// TwinCAT 3 PLC project Welding_Robot_Control_Test
// ProgramVersion: 3.1.4020.4
// libraries:
//   Tc2_MC2, * (Beckhoff Automation GmbH)
//   Tc2_Standard, * (Beckhoff Automation GmbH)
//   Tc2_System, * (Beckhoff Automation GmbH)
//   Tc3_Module, * (Beckhoff Automation GmbH)
//   VisuDialogs, * (System)
// project tree:
//   DUTs/Axis/ Axis.TcPOU (not stored)
//   DUTs/Delay/ Delay.TcPOU (not stored)
//   DUTs/Filter_Current/ E_TcMatSimDataAreaType_1.TcDUT (not stored), FB_Filter_Current_Hexapod_Robot.TcPOU (not stored), FB_TcMatSimObject_1.TcPOU (not stored), ST_Filter_Current_Hexapod_Robot_InitData.TcDUT (not stored), ST_Filter_Current_Hexapod_Robot_Input.TcDUT (not stored), ST_Filter_Current_Hexapod_Robot_Output.TcDUT (not stored), ST_TcMatSimObjectDataAreaInfo_1.TcDUT (not stored)
//   DUTs/Hexapod_Leg/ Hexapod_Leg.TcPOU (not stored)
//   DUTs/Mapping/ Hexapod_Robot_Mapping.TcPOU (not stored)
//   DUTs/Robot_Simulink/ E_TcMatSimDataAreaType.TcDUT, FB_TcMatSimObject.TcPOU, FB_Welding_Control_Circle_86s.TcPOU, ST_TcMatSimObjectDataAreaInfo.TcDUT, ST_Welding_Control_Circle_86s_InitData.TcDUT, ST_Welding_Control_Circle_86s_Input.TcDUT, ST_Welding_Control_Circle_86s_Output.TcDUT
//   / GlobalTextList.TcGTLO, HexRobot_Task.TcTTO, PlcTask.TcTTO, Welding_Arm_Task.TcTTO, 视图管理器.TcVMO (not stored)
//   GVLs/ GVL.TcGVL
//   POUs/ Hexapod_Robot.TcPOU, Welding_Arm.TcPOU, Welding_Robot.TcPOU
//   VISUs/ Visu_Home.TcVIS, Visu_SimulinkMove.TcVIS, Visu_Power.TcVIS, Visu_Reset.TcVIS, Visu_Stand.TcVIS (not stored)

CONFIGURATION Welding_Robot_Control_Test
    RESOURCE PLC ON TwinCAT3
        TASK HexRobot_Task(INTERVAL := T#1ms, PRIORITY := 21);
        TASK PlcTask(INTERVAL := T#1ms, PRIORITY := 20);
        TASK Welding_Arm_Task(INTERVAL := T#1ms, PRIORITY := 22);
        PROGRAM Hexapod_Robot WITH HexRobot_Task : Hexapod_Robot;
        PROGRAM Welding_Robot WITH PlcTask : Welding_Robot;
        PROGRAM Welding_Arm WITH Welding_Arm_Task : Welding_Arm;
    END_RESOURCE
END_CONFIGURATION

// ---- DUTs/Robot_Simulink/E_TcMatSimDataAreaType.TcDUT
TYPE E_TcMatSimDataAreaType :
(
	NotSpecified := 0,
	Standard,
	InputSrc,
	InputDst,
	OutputSrc,
	OutputDst,
	InternalDa,
	MArea,
	RetainDa
);
END_TYPE

// ---- DUTs/Robot_Simulink/ST_TcMatSimObjectDataAreaInfo.TcDUT
TYPE ST_TcMatSimObjectDataAreaInfo :
STRUCT
	pPlcVar: PVOID;
	pModuleProcImg: PVOID;
	nSize: UDINT;
	nDataAreaId: UDINT;
	eDataAreaType: E_TcMatSimDataAreaType;
END_STRUCT
END_TYPE

// ---- DUTs/Robot_Simulink/ST_Welding_Control_Circle_86s_InitData.TcDUT
{attribute 'pack_mode' := '4'}
TYPE ST_Welding_Control_Circle_86s_InitData :
STRUCT
	Header: TComInitDataHdr;
	CallByHdr: TComInitDataElmHdr;
	CallBy: TctModuleCallByType;
	ExecutionSequenceHdr: TComInitDataElmHdr;
	ExecutionSequence: TctModuleExecutionSequenceType;
	StepSizeHdr: TComInitDataElmHdr;
	StepSize: TctStepSizeType;
	ExecuteModelCodeHdr: TComInitDataElmHdr;
	ExecuteModelCode: BOOL;
	ContextInfoArr_0_TaskOidHdr: TComInitDataElmHdr;
	ContextInfoArr_0_TaskOid: OTCID;
	ContextInfoArr_0_TaskPriorityHdr: TComInitDataElmHdr;
	ContextInfoArr_0_TaskPriority: UDINT;
	ContextInfoArr_0_TaskCycleTimeNsHdr: TComInitDataElmHdr;
	ContextInfoArr_0_TaskCycleTimeNs: UDINT;
	ContextInfoArr_0_TaskPortHdr: TComInitDataElmHdr;
	ContextInfoArr_0_TaskPort: UINT;
	ContextInfoArr_0_TaskSortOrderHdr: TComInitDataElmHdr;
	ContextInfoArr_0_TaskSortOrder: UDINT;
END_STRUCT
END_TYPE

// ---- DUTs/Robot_Simulink/ST_Welding_Control_Circle_86s_Input.TcDUT
TYPE ST_Welding_Control_Circle_86s_Input :
STRUCT
	t: LREAL;
END_STRUCT
END_TYPE

// ---- DUTs/Robot_Simulink/ST_Welding_Control_Circle_86s_Output.TcDUT
TYPE ST_Welding_Control_Circle_86s_Output :
STRUCT
	Disp_P: matrix_18_real_T;
END_STRUCT
END_TYPE

// ---- GVLs/GVL.TcGVL
VAR_GLOBAL
	Power_Execute 		: BOOL;							// 上电使能控制信号
	Home_Execute		: BOOL;							// 设置零点程序使能
	Reset_Execute		: BOOL;							// 电机驱动重置动作发生使能
	ExSetPoint_Execute	: BOOL;							// 机器人外部信号发生使能
	
	// ====================Simulink模块相关=====================
	Robot_Simulink		: FB_Welding_Control_Circle_86s(oid:=16#01010020);	// Simulink模型定义
	T_ALL				: LREAL:=100;						// Simulink模型运动总时长
	t_Interval			: LREAL:=0.001;						// 取样时间间隔，默认为1ms
	t					: LREAL:=0;							// 取样当前时间变量，以0为起点
	
	Filter_Current  : FB_Filter_Current_Hexapod_Robot(oid:=16#01010030);

END_VAR

// ---- POUs/Hexapod_Robot.TcPOU
PROGRAM Hexapod_Robot
VAR
// =======================NC轴变量==========================
	//Leg_Robot			: ARRAY[1..6] OF Hexapod_Leg;	// 定义六足的腿
	Axis_Robot			: ARRAY[1..18] OF Axis;			// 定义六足轴参量(可以调整数据上限来调整电机数目)
	//Axis_Delay			: Delay;						// 延迟程序
	Leg_Number			: INT;							// 定义机器人腿数
	Axis_Number 		: INT;							// 定义轴数目
	
	// ===================模块动作信号(按动作先后排列)==========
	Axis_Power			: ARRAY[1..18] OF BOOL;			// 单电机使能
	Robot_Power			: BOOL;							// 机器人所有电机使能
	
	Leg_Home_Set		: ARRAY[1..6] OF BOOL;	
	Axis_Home_Set		: ARRAY[1..18] OF BOOL;			// 单电机设定零点信号
	Robot_Home_Set		: BOOL;							// 机器人所有电机设定零点信号
	
	Move_Execute		: BOOL;							// 绝对运动使能信号
	Robot_Stand_Execute	: BOOL;							// 机器人站立程序使能	
	Axis_Absolute_Eable	: ARRAY[1..18] OF BOOL;			// 单电机绝对运动使能信号
	Robot_Absolute_Eable: ARRAY[1..18] OF BOOL;			// 机器人站立使能信号
	Axis_Move_Position	: ARRAY[1..18] OF LREAL;		// 电机绝对运动位置			
	
	ExtSetPointEnable	: BOOL;							// 外部信号发生信号
	ExtSetPointDisable	: BOOL;							// 外部信号结束信号
	
	Axis_Reset			: ARRAY[1..18] OF BOOL;			// 单电机驱动重置信号使能
	Robot_Reset			: BOOL;							// 机器人整体电机驱动重置
	Axis_ResetDone		: ARRAY[1..18] OF BOOL;			// 单电机驱动重置完成
	
	// ===================状态监测变量=======================
	Power_Status	: ARRAY[1..18] OF BOOL;				// 上电监测信号
	Leg_Home_Done	: ARRAY[1..6] OF BOOL;
	Home_Done		: ARRAY[1..18] OF BOOL;				// 找零监测信号
	MoveAbsoluteDone: ARRAY[1..18] OF BOOL;				// 电机运动监测信号
	
	Robot_Error		: BOOL;								// 机器人电机错误信号
	Axis_Error		: ARRAY[1..18] OF BOOL;				// 电机错误监测信号
	Axis_ErrorID	: ARRAY[1..18] OF UDINT;			// 电机错误号码监测信号
	
	Axis_ActPostion	: ARRAY[1..18] OF LREAL;			// 电机轴实际位置
	Difference_Position	: ARRAY[1..18] OF LREAL;		// 实际位置与输入位置差值
	
	// =======================模块中间变量======================
	//HomeDone_Number	: LREAL :=0;					//完成找零的轴数
	//ExSetPoint_Position	: ARRAY[1..18] OF LREAL;		// 外部信号位置
	//t					: LREAL :=0;
	
	// =======================驱动器信号监测====================
	Current_Turque_Value  AT%IW0 : ARRAY[1..18] OF INT ;	//电流、力矩相关值
	Max_Turque_Value 	: INT ;							// 设置最大力矩边界值
	
	// ====================Simulink模块相关=====================
	Mapping				: Hexapod_Robot_Mapping;			// 变量映射	
	Model_Position		: ARRAY[1..18] OF LREAL;			// Simulink中各个腿的位置
	ExSetPoint_Position	: ARRAY[1..18] OF LREAL;			// 外部信号位置		
	Home_Position 		: ARRAY[1..18] OF LREAL;			// Home结束后的位移值
	
	Current_Turque_Filter  : ARRAY[1..18] OF LREAL;			// 滤波后的电流值
 
END_VAR

// =======================子程序使能(永久运行)===================
Variable_Monitor();			// 变量监测子程序使能
Logic_Control();			// 逻辑控制子程序使能
Variable_Set();				// 各动作速度子程序使能
SetGenerator();				// 外部信号发生子程序使能
Leg_Action();				// 单腿运动子程序使能
Robot_Action();				// 机器人整体运动子程序使能

// =====================电机驱动重置=============================
IF Reset_Execute THEN
	FOR Axis_Number := 1 TO 18 {BY 1} DO
		Axis_Robot[Axis_Number].Reset(Drive_Reset:= Axis_Reset[Axis_Number]);
	END_FOR
END_IF

// =======================电机上电===============================
IF Power_Execute THEN
	Filter_Current.Execute();
	FOR Axis_Number := 1 TO 18 {BY 1} DO
		Axis_Robot[Axis_Number].Power(Axis_Enable:= Axis_Power[Axis_Number]);
	END_FOR
END_IF

// =======================找零程序===============================
IF Home_Execute THEN
	Robot_Simulink.Execute();	// Simulink模型使能，用来为找零后的电机提供初始位移
	FOR Axis_Number := 1 TO 18 {BY 1} DO
		Axis_Robot[Axis_Number].Home(Drive_Home:= Axis_Home_Set[Axis_Number]);
	END_FOR
END_IF

// =======================站立程序===============================
IF Move_Execute THEN
	FOR Axis_Number := 1 TO 18 {BY 1} DO
		Axis_Robot[Axis_Number].Move_Absolute(	Drive_Move_Absolute:= Axis_Absolute_Eable[Axis_Number], 
												Absolute_Position:= Axis_Move_Position[Axis_Number]);
	END_FOR
END_IF
	
// =======================外部信号运动程序=======================
IF ExSetPoint_Execute THEN
	//SetGenerator();			// 使能外部信号发生子程序
	Robot_Simulink.Execute();	// Simulink模型使能
	FOR Axis_Number := 1 TO 18 {BY 1} DO
		Axis_Robot[Axis_Number].ExtSetPoint(Drive_ExtSetPointEnable:= ExtSetPointEnable, 
											Drive_ExtSetPointDisable:= ExtSetPointDisable, 
											ExSetPosition:= ExSetPoint_Position[Axis_Number]);
	END_FOR
END_IF

ACTION Leg_Action:
// ===================机器人单挑腿找零程序====================
IF Home_Execute THEN
	FOR Leg_Number := 1 TO 6 {BY 1} DO
		IF Leg_Home_Set[Leg_Number] THEN		// 在可视化中，Leg_Home_Set为点动
			Axis_Home_Set[1+(Leg_Number-1)*3] := Leg_Home_Set[Leg_Number];
			Axis_Home_Set[2+(Leg_Number-1)*3] := Leg_Home_Set[Leg_Number];
			Axis_Home_Set[3+(Leg_Number-1)*3] := Leg_Home_Set[Leg_Number];
		ELSIF Home_Done[1+(Leg_Number-1)*3] AND Axis_Home_Set[2+(Leg_Number-1)*3] AND Axis_Home_Set[3+(Leg_Number-1)*3] THEN
			Leg_Home_Set[Leg_Number] := FALSE; 
		END_IF
	END_FOR
END_IF
END_ACTION

ACTION Logic_Control:
// =======================控制逻辑区==========================
// 保证所有的动作拥有合理的先后顺序，优化控制逻辑
// 也防止出现两个或两个以上动作同时进行的情况，保证控制安全

// ===================电机驱动重置逻辑========================
//FOR Axis_Number := 1 TO 18 {BY 1} DO
IF Axis_Error[1] OR Axis_Error[2] OR Axis_Error[3] OR Axis_Error[4] OR Axis_Error[5] OR Axis_Error[6]
	 OR Axis_Error[7] OR Axis_Error[8] OR Axis_Error[9] OR Axis_Error[10] OR Axis_Error[11] OR Axis_Error[12]
		OR Axis_Error[13] OR Axis_Error[14] OR Axis_Error[15] OR Axis_Error[16] OR Axis_Error[17] OR Axis_Error[18]
THEN
	Robot_Error := TRUE;
ELSE
	Robot_Error := FALSE;
END_IF
//END_FOR

IF Robot_Error THEN
	Reset_Execute := TRUE;
ELSIF NOT Robot_Error AND NOT Welding_Arm.Arm_Error THEN
	Reset_Execute := FALSE;
ELSIF NOT Reset_Execute THEN
	Axis_Reset[Axis_Number] := FALSE;
	Axis_Robot[Axis_Number].Reset(Drive_Reset:= Axis_Reset[Axis_Number]);
END_IF

// =====================上电程序逻辑==========================
IF NOT Power_Execute THEN
	FOR Axis_Number := 1 TO 18 {BY 1} DO
		Axis_Power[Axis_Number] := FALSE;
		Axis_Robot[Axis_Number].Power(Axis_Enable:= Axis_Power[Axis_Number]);
	END_FOR
END_IF

// =====================找零程序逻辑==========================
IF Home_Execute THEN
	FOR Axis_Number := 1 TO 18 {BY 1} DO
		IF Home_Done[Axis_Number] THEN			// 	丝杠到达零点位置后，单电j机标零使能位关闭			
			Axis_Home_Set[Axis_Number] :=0;	
			Axis_Robot[Axis_Number].Home(Drive_Home:= Axis_Home_Set[Axis_Number]);
		END_IF
	END_FOR
	Move_Execute :=0;							// 设定零点时，不能进行其他运动
	ExSetPoint_Execute :=0;
ELSIF NOT Home_Execute THEN
	FOR Axis_Number := 1 TO 18 {BY 1} DO
		//Axis_Start_Back[Axis_Number] :=0;
		Axis_Home_Set[Axis_Number] := 0;
	END_FOR
END_IF

// =====================机器人站立逻辑==========================
IF Move_Execute THEN
	//Absolute_Eable := TRUE;
	Home_Execute := FALSE;						// 站立运动使能时，机器人调零必须结束
	ExSetPoint_Execute :=0;						// 站立运动时，不能进行其他运动
	FOR Axis_Number := 1 TO 18 {BY 1} DO
		IF MoveAbsoluteDone[Axis_Number] THEN	// 	丝杠到达设定位置后，单电机绝对运动使能位关闭
			Axis_Absolute_Eable[Axis_Number] := FALSE;
		END_IF
	END_FOR
ELSIF NOT Move_Execute THEN						// 站立运动不使能,轴不能运动
	FOR Axis_Number := 1 TO 18 {BY 1} DO
		Axis_Absolute_Eable[Axis_Number] := FALSE;
		Axis_Robot[Axis_Number].Move_Absolute(	Drive_Move_Absolute:= Axis_Absolute_Eable[Axis_Number], 
												Absolute_Position:= Axis_Move_Position[Axis_Number]);
	END_FOR
END_IF

// =====================外部信号发生逻辑========================
IF ExSetPoint_Execute THEN
	Home_Execute := FALSE;						// 外部信号发生使能时，机器人调零必须结束
	Move_Execute :=0;							// 外部信号发生时，不能进行其他运动
ELSIF NOT ExSetPoint_Execute THEN
	ExtSetPointEnable := 0;						// 外部信号发生不使能时，外部信号不能进入程序
	ExtSetPointDisable :=0;
ELSIF ExtSetPointDisable THEN
	ExtSetPointEnable :=0;						// 外部信号发生停止与外部信号发生开始不能同时进行
END_IF
END_ACTION

ACTION Robot_Action:
// =================机器人整体运动命令区======================
// 六足所有电机整体控制

// ====================机器人驱动重置=========================
IF Robot_Reset THEN
	IF Reset_Execute THEN
		Axis_Reset[Axis_Number] := TRUE;
		FOR Axis_Number := 1 TO 18 {BY 1} DO
			Axis_Robot[Axis_Number].Reset(Drive_Reset:= Axis_Reset[Axis_Number]);
		END_FOR
	END_IF
END_IF	

// ===================机器人所有电机上电======================
IF Robot_Power THEN	
	IF Power_Execute THEN
		FOR Axis_Number := 1 TO 18 {BY 1} DO
			Axis_Power[Axis_Number] := TRUE ;
		END_FOR
	END_IF
END_IF
	
// ===================机器人找零程序=======================
IF Robot_Home_Set THEN				// 标零程序
	//Robot_Start_Back := FALSE;
	IF Home_Execute THEN
		Leg_Home_Set[3] := Leg_Home_Set[5] := Leg_Home_Set[1];	// 在整机调零时，1\3\5三条腿同时调零；
		Leg_Home_Set[4] := Leg_Home_Set[6] := Leg_Home_Set[2];	// 在整机调零时，2\4\6三条腿同时调零；
	ELSIF NOT Home_Execute THEN
		FOR Leg_Number := 1 TO 6 {BY 1} DO
			Leg_Home_Set[Leg_Number] := FALSE;
		END_FOR
	END_IF
ELSIF NOT Robot_Home_Set AND NOT Home_Execute THEN
	FOR Axis_Number := 1 TO 18 {BY 1} DO
	Axis_Home_Set[Axis_Number] := FALSE;
	END_FOR
END_IF

// =====================站立程序===============================
IF Robot_Stand_Execute THEN
	IF Move_Execute THEN
		FOR Axis_Number := 1 TO 18 {BY 1} DO
			IF MoveAbsoluteDone[Axis_Number] THEN		// 	丝杠到达设定位置后，单电机绝对运动使能位关闭
				Axis_Absolute_Eable[Axis_Number] := FALSE;
			ELSE
				Axis_Absolute_Eable[Axis_Number] := TRUE;
			END_IF
		END_FOR
	END_IF
ELSIF NOT Robot_Stand_Execute AND NOT Move_Execute THEN 
	FOR Axis_Number := 1 TO 18 {BY 1} DO
		Axis_Absolute_Eable[Axis_Number] := FALSE;
	END_FOR
END_IF

// ======================外部信号发生=========================
IF ExtSetPointEnable THEN	
	//FOR Axis_Number := 1 TO 2 {BY 1} DO
	t := t + t_Interval;
	ExtSetPointDisable := FALSE;
	//END_FOR
END_IF

IF t=0 THEN
	FOR Axis_Number := 1 TO 18 {BY 1} DO
		Home_Position[Axis_Number] := Axis_ActPostion[Axis_Number];
	END_FOR
ELSIF t>=T_ALL THEN
	ExtSetPointEnable := FALSE;
	t:=0;
	ExtSetPointDisable := TRUE;
END_IF
END_ACTION

ACTION SetGenerator:
// ====================外部信号发生测试区=====================
// 用来测试外部信号发生功能和电机相关参数

// =================外部信号正弦信号发生======================
(*IF ExtSetPointEnable THEN
	FOR Axis_Number := 1 TO 18 {BY 1} DO
		ExSetPoint_Position[Axis_Number]:=10*SIN(2*3.14*t);
		t := t+0.001;
	END_FOR
END_IF

// =================外部信号停止逻辑判断=======================
//IF Axis_Robot[Axis_Number].State_ExtSetPiontDone THEN
IF t>=20 THEN
	ExtSetPointEnable := FALSE;
	t:=0;
	ExtSetPointDisable := TRUE;
END_IF
//END_IF*)
END_ACTION

ACTION Variable_Monitor:
// =====================关键数据信号监测======================

// ==============最大力矩设置区(边界控制条件)=================
FOR Axis_Number := 1 TO 18 {BY 1} DO
	Axis_Robot[Axis_Number].Max_Turque_Value := Max_Turque_Value;
END_FOR

// =======================力矩检测区==========================
FOR Axis_Number := 1 TO 18 {BY 1} DO
	Axis_Robot[Axis_Number].Current_Turque_Value := Current_Turque_Value[Axis_Number];
END_FOR

// ====================轴实际位置检测区=======================
FOR Axis_Number := 1 TO 18 {BY 1} DO
	Axis_ActPostion[Axis_Number] := Axis_Robot[Axis_Number].ActPosition;
END_FOR

// =======================上电状态检测区======================
FOR Axis_Number := 1 TO 18 {BY 1} DO
	Power_Status[Axis_Number] := Axis_Robot[Axis_Number].State_PowerStatus;
END_FOR

// =======================找零状态检测区======================
FOR Axis_Number := 1 TO 18 {BY 1} DO
	Home_Done[Axis_Number] := Axis_Robot[Axis_Number].State_HomeDone;
END_FOR

(*FOR Leg_Number := 1 TO 6 {BY 1} DO
	Leg_Home_Done[Leg_Number] := Leg_Robot[Axis_Number].State_HomeDone;
END_FOR*)

// ===================电机绝对运动状态检测区==================
FOR Axis_Number := 1 TO 18 {BY 1} DO
	MoveAbsoluteDone[Axis_Number] := Axis_Robot[Axis_Number].State_MoveAbsoluteDone;
END_FOR

// =======================电机错误检测区======================
FOR Axis_Number := 1 TO 18 {BY 1} DO
	Axis_Error[Axis_Number] := Axis_Robot[Axis_Number].Axis_Error;
	Axis_ErrorID[Axis_Number] := Axis_Robot[Axis_Number].Axis_ErrorID;
END_FOR

// ==============实际运动位移和输入位移差值检测区==============
FOR Axis_Number := 1 TO 18 {BY 1} DO
	Difference_Position[Axis_Number] := Axis_ActPostion[Axis_Number]- Mapping.Controller_Leg_Position[Axis_Number]; 
END_FOR
END_ACTION

ACTION Variable_Set:
// =======================速度规定区==========================
FOR Axis_Number := 1 TO 18 {BY 1} DO						//此时每一个电机的速度都是一样的
	Axis_Robot[Axis_Number].Home_Velocity 	:= 20;			//找零速度(Axis_Jog中的速度)
	Axis_Robot[Axis_Number].Move_Relative_Velocity	:=30;	//相对运动速度
END_FOR
IF Home_Execute THEN
	//IF Robot_Home_Set THEN
		Axis_Robot[1].Move_Absolute_Velocity :=17; Axis_Robot[3].Move_Absolute_Velocity :=17; Axis_Robot[4].Move_Absolute_Velocity :=16.74;
		Axis_Robot[6].Move_Absolute_Velocity :=16.74; Axis_Robot[7].Move_Absolute_Velocity :=17.3; Axis_Robot[9].Move_Absolute_Velocity :=17.3;
		Axis_Robot[10].Move_Absolute_Velocity :=16.95; Axis_Robot[12].Move_Absolute_Velocity :=16.95; Axis_Robot[13].Move_Absolute_Velocity :=17;
		Axis_Robot[15].Move_Absolute_Velocity :=17; Axis_Robot[16].Move_Absolute_Velocity :=17; Axis_Robot[18].Move_Absolute_Velocity :=17;
		Axis_Robot[2].Move_Absolute_Velocity :=20; Axis_Robot[5].Move_Absolute_Velocity :=20; Axis_Robot[8].Move_Absolute_Velocity :=20;
		Axis_Robot[11].Move_Absolute_Velocity :=20; Axis_Robot[14].Move_Absolute_Velocity :=20; Axis_Robot[17].Move_Absolute_Velocity :=20;
	//ELSIF NOT Robot_Home_Set THEN
		//FOR Axis_Number := 1 TO 18 {BY 1} DO
			//Axis_Robot[Axis_Number].Move_Absolute_Velocity	:=10;
		//END_FOR
	//END_IF
ELSE
	FOR Axis_Number := 1 TO 18 {BY 1} DO
			Axis_Robot[Axis_Number].Move_Absolute_Velocity	:=10;
	END_FOR
END_IF
	

// =======================位置规定区==========================
FOR Axis_Number := 1 TO 18 {BY 1} DO
	Axis_Move_Position[Axis_Number] := 160;
END_FOR

// =====================最大力矩规定区========================
Max_Turque_Value := 1300;

// ===============电机设置零点后到达位置规定区================
(*Axis_Robot[1].Home_Absolute_Position := 73.7632; Axis_Robot[3].Home_Absolute_Position := 73.7632; Axis_Robot[4].Home_Absolute_Position := 73.7632;
Axis_Robot[6].Home_Absolute_Position := 73.7632; Axis_Robot[7].Home_Absolute_Position := 73.7632; Axis_Robot[9].Home_Absolute_Position := 73.7632;
Axis_Robot[10].Home_Absolute_Position := 73.7632; Axis_Robot[12].Home_Absolute_Position := 73.7632; Axis_Robot[13].Home_Absolute_Position := 73.7632;
Axis_Robot[15].Home_Absolute_Position := 73.7632; Axis_Robot[16].Home_Absolute_Position := 73.7632; Axis_Robot[18].Home_Absolute_Position := 73.7632;
Axis_Robot[2].Home_Absolute_Position := 83.7506; Axis_Robot[5].Home_Absolute_Position := 83.7506; Axis_Robot[8].Home_Absolute_Position := 83.7506;
Axis_Robot[11].Home_Absolute_Position := 83.7506; Axis_Robot[14].Home_Absolute_Position := 83.7506; Axis_Robot[17].Home_Absolute_Position := 83.7506;*)
(*Axis_Robot[1].Home_Absolute_Position := 138; Axis_Robot[3].Home_Absolute_Position := 138; Axis_Robot[4].Home_Absolute_Position := 138;
Axis_Robot[6].Home_Absolute_Position := 138; Axis_Robot[7].Home_Absolute_Position := 138; Axis_Robot[9].Home_Absolute_Position := 138;
Axis_Robot[10].Home_Absolute_Position := 138; Axis_Robot[12].Home_Absolute_Position := 138; Axis_Robot[13].Home_Absolute_Position := 138;
Axis_Robot[15].Home_Absolute_Position := 138; Axis_Robot[16].Home_Absolute_Position := 138; Axis_Robot[18].Home_Absolute_Position := 138;
Axis_Robot[2].Home_Absolute_Position := 149; Axis_Robot[5].Home_Absolute_Position := 149; Axis_Robot[8].Home_Absolute_Position := 149;
Axis_Robot[11].Home_Absolute_Position := 149; Axis_Robot[14].Home_Absolute_Position := 149; Axis_Robot[17].Home_Absolute_Position := 149;*)
FOR Axis_Number := 1 TO 18 {BY 1} DO
	Axis_Robot[Axis_Number].Home_Absolute_Position := Mapping.Controller_Leg_Position[Axis_Number];
END_FOR

// ===================外部信号发生电机位置输入值================
FOR Axis_Number := 1 TO 18 {BY 1} DO
	ExSetPoint_Position[Axis_Number]:= Mapping.Controller_Leg_Position[Axis_Number];
END_FOR

// ===================电机和腿映射关系========================
//FOR Leg_Number := 1 TO 6 {BY 1} DO
(*Leg_Robot[1](Axis1:= Axis_Robot[1], Axis2:= Axis_Robot[2], Axis3:= Axis_Robot[3]);
Leg_Robot[2](Axis1:= Axis_Robot[4], Axis2:= Axis_Robot[5], Axis3:= Axis_Robot[6]);
Leg_Robot[3](Axis1:= Axis_Robot[7], Axis2:= Axis_Robot[8], Axis3:= Axis_Robot[9]);
Leg_Robot[4](Axis1:= Axis_Robot[10], Axis2:= Axis_Robot[11], Axis3:= Axis_Robot[12]);
Leg_Robot[5](Axis1:= Axis_Robot[13], Axis2:= Axis_Robot[14], Axis3:= Axis_Robot[15]);
Leg_Robot[6](Axis1:= Axis_Robot[16], Axis2:= Axis_Robot[17], Axis3:= Axis_Robot[18]);*)
//END_FOR

// ===================程序与模型的变量链接===================
Mapping(Model_Leg_Position:= Model_Position);				// 映射运动学模型中腿编号和控制模型中的电机编号
Robot_Simulink.stInput.t := t;								// 采样时间t与Simulink模型中的采样时间链接
Model_Position := Robot_Simulink.stOutput.Disp_P;			// Simulink中的电机输出位移输入到控制模型
FOR Axis_Number := 1 TO 18 {BY 1} DO
	Filter_Current.stInput.Current_Motor[Axis_Number-1] := Current_Turque_Value[Axis_Number];
END_FOR	
Current_Turque_Filter := Filter_Current.stOutput.Current_Monitor;
END_ACTION

END_PROGRAM

// ---- POUs/Welding_Arm.TcPOU
PROGRAM Welding_Arm
VAR
	Axis_Arm			: ARRAY[1..3] OF Axis;				// 定义焊接臂上电机
	Axis_Number 		: INT;								// 定义轴数目
	
	// ===================模块动作信号(按动作先后排列)==========
	Axis_Power			: ARRAY[1..3] OF BOOL;				// 单电机使能
	Arm_Power			: BOOL;								// 机器人所有电机使能
	
	Axis_Home_Set		: ARRAY[1..3] OF BOOL;				// 单电机设定零点信号
	Arm_Home_Set		: BOOL;								// 机器人所有电机设定零点信号		
	
	Axis_Reset			: ARRAY[1..3] OF BOOL;				// 单电机驱动重置信号使能
	Robot_Reset			: BOOL;								// 机器人整体电机驱动重置
	Axis_ResetDone		: ARRAY[1..3] OF BOOL;				// 单电机驱动重置完成
	
	ExtSetPointEnable	: BOOL;								// 外部信号发生信号
	ExtSetPointDisable	: BOOL;								// 外部信号结束信号
	
	// ===================状态监测变量=======================
	Power_Status	: ARRAY[1..3] OF BOOL;					// 上电监测信号
	Home_Done		: ARRAY[1..3] OF BOOL;					// 找零监测信号
	MoveAbsoluteDone: ARRAY[1..3] OF BOOL;					// 电机运动监测信号
	
	Arm_Error		: BOOL;									// 焊接臂电机错误信号
	Axis_Error		: ARRAY[1..3] OF BOOL;					// 电机错误监测信号
	Axis_ErrorID	: ARRAY[1..3] OF UDINT;					// 电机错误号码监测信号
	
	Axis_ActPostion	: ARRAY[1..3] OF LREAL;					// 电机轴实际位置
	Difference_Position	: ARRAY[1..3] OF LREAL;				// 实际位置与输入位置差值
	
	// =======================驱动器信号监测====================
	Current_Turque_Value  AT%IW0 : ARRAY[1..3] OF INT ;		//电流、力矩相关值
	Max_Turque_Value 	: INT ;								// 设置最大力矩边界值
	
	// ====================Simulink模块相关=====================	
	ExSetPoint_Position	: ARRAY[1..3] OF LREAL;			// 外部信号位置	
	Home_Position 		: ARRAY[1..3] OF LREAL;				// Home结束后的位移值
	Model_Position		: ARRAY[1..3] OF LREAL;			// Simulink中各个腿的位置
	Current_Turque_Filter  : ARRAY[1..3] OF LREAL;			// 滤波后的电流值
END_VAR

// =======================子程序使能(永久运行)===================
Variable_Monitor();			// 变量监测子程序使能
Logic_Control();			// 逻辑控制子程序使能
Variable_Set();				// 各动作速度子程序使能

// =====================电机驱动重置=============================
IF Reset_Execute THEN
	FOR Axis_Number := 1 TO 3 {BY 1} DO
		Axis_Arm[Axis_Number].Reset(Drive_Reset:= Axis_Reset[Axis_Number]);
	END_FOR
END_IF

// =======================电机上电===============================
IF Power_Execute THEN
	Filter_Current.Execute();
	FOR Axis_Number := 1 TO 3 {BY 1} DO
		Axis_Arm[Axis_Number].Power(Axis_Enable:= Axis_Power[Axis_Number]);
	END_FOR
END_IF

// =======================找零程序===============================
IF Home_Execute THEN
	FOR Axis_Number := 1 TO 3 {BY 1} DO
		Axis_Arm[Axis_Number].Home(Drive_Home:= Axis_Home_Set[Axis_Number]);
	END_FOR
END_IF
	
// =======================外部信号运动程序=======================
IF ExSetPoint_Execute THEN
	FOR Axis_Number := 1 TO 3 {BY 1} DO
		Axis_Arm[Axis_Number].ExtSetPoint(	Drive_ExtSetPointEnable:= ExtSetPointEnable, 
											Drive_ExtSetPointDisable:= ExtSetPointDisable, 
											ExSetPosition:= ExSetPoint_Position[Axis_Number]);
	END_FOR
END_IF

ACTION Logic_Control:
// =======================控制逻辑区==========================
// 保证所有的动作拥有合理的先后顺序，优化控制逻辑
// 也防止出现两个或两个以上动作同时进行的情况，保证控制安全

// ===================电机驱动重置逻辑========================
IF Axis_Error[1] OR Axis_Error[2] OR Axis_Error[3] THEN
	Arm_Error := TRUE;
ELSE
	Arm_Error := FALSE;
END_IF
//END_FOR

IF Arm_Error THEN
	Reset_Execute := TRUE;
ELSIF NOT Arm_Error AND NOT Hexapod_Robot.Robot_Error THEN
	Reset_Execute := FALSE;
ELSIF NOT Reset_Execute THEN
	Axis_Reset[Axis_Number] := FALSE;
	Axis_Arm[Axis_Number].Reset(Drive_Reset:= Axis_Reset[Axis_Number]);
END_IF

// =====================上电程序逻辑==========================
IF NOT Power_Execute THEN
	FOR Axis_Number := 1 TO 3 {BY 1} DO
		Axis_Power[Axis_Number] := FALSE;
		Axis_Arm[Axis_Number].Power(Axis_Enable:= Axis_Power[Axis_Number]);
	END_FOR
END_IF

// =====================找零程序逻辑==========================
IF Home_Execute THEN
	FOR Axis_Number := 1 TO 3 {BY 1} DO
		IF Home_Done[Axis_Number] THEN			// 	丝杠到达零点位置后，单电机标零使能位关闭			
			Axis_Home_Set[Axis_Number] :=0;	
			Axis_Arm[Axis_Number].Home(Drive_Home:= Axis_Home_Set[Axis_Number]);
		END_IF
	END_FOR
	ExSetPoint_Execute :=0;
ELSIF NOT Home_Execute THEN
	FOR Axis_Number := 1 TO 3 {BY 1} DO
		//Axis_Start_Back[Axis_Number] :=0;
		Axis_Home_Set[Axis_Number] := 0;
	END_FOR
END_IF

// =====================外部信号发生逻辑========================
IF ExSetPoint_Execute THEN
	Home_Execute := FALSE;						// 外部信号发生使能时，机器人调零必须结束
ELSIF NOT ExSetPoint_Execute THEN
	ExtSetPointEnable := 0;						// 外部信号发生不使能时，外部信号不能进入程序
	ExtSetPointDisable :=0;
ELSIF ExtSetPointDisable THEN
	ExtSetPointEnable :=0;						// 外部信号发生停止与外部信号发生开始不能同时进行
END_IF

IF ExtSetPointEnable THEN	
	//FOR Axis_Number := 1 TO 2 {BY 1} DO
	t := t + t_Interval;
	ExtSetPointDisable := FALSE;
	//END_FOR
END_IF

IF t=0 THEN
	FOR Axis_Number := 1 TO 3 {BY 1} DO
		Home_Position[Axis_Number] := Axis_ActPostion[Axis_Number];
	END_FOR
ELSIF t>=T_ALL THEN
	ExtSetPointEnable := FALSE;
	t:=0;
	ExtSetPointDisable := TRUE;
END_IF
END_ACTION

ACTION Variable_Monitor:
// =====================关键数据信号监测======================

// ==============最大力矩设置区(边界控制条件)=================
FOR Axis_Number := 1 TO 3 {BY 1} DO
	Axis_Arm[Axis_Number].Max_Turque_Value := Max_Turque_Value;
END_FOR

// =======================力矩检测区==========================
FOR Axis_Number := 1 TO 3 {BY 1} DO
	Axis_Arm[Axis_Number].Current_Turque_Value := Current_Turque_Value[Axis_Number];
END_FOR

// ====================轴实际位置检测区=======================
FOR Axis_Number := 1 TO 3 {BY 1} DO
	Axis_ActPostion[Axis_Number] := Axis_Arm[Axis_Number].ActPosition;
END_FOR

// =======================上电状态检测区======================
FOR Axis_Number := 1 TO 3 {BY 1} DO
	Power_Status[Axis_Number] := Axis_Arm[Axis_Number].State_PowerStatus;
END_FOR

// =======================找零状态检测区======================
FOR Axis_Number := 1 TO 3 {BY 1} DO
	Home_Done[Axis_Number] := Axis_Arm[Axis_Number].State_HomeDone;
END_FOR

// ===================电机绝对运动状态检测区==================
FOR Axis_Number := 1 TO 3 {BY 1} DO
	MoveAbsoluteDone[Axis_Number] := Axis_Arm[Axis_Number].State_MoveAbsoluteDone;
END_FOR

// =======================电机错误检测区======================
FOR Axis_Number := 1 TO 3 {BY 1} DO
	Axis_Error[Axis_Number] := Axis_Arm[Axis_Number].Axis_Error;
	Axis_ErrorID[Axis_Number] := Axis_Arm[Axis_Number].Axis_ErrorID;
END_FOR
END_ACTION

ACTION Variable_Set:
// =======================速度规定区==========================
FOR Axis_Number := 1 TO 3 {BY 1} DO						//此时每一个电机的速度都是一样的
	Axis_Arm[Axis_Number].Home_Velocity 	:= 20;			//找零速度(Axis_Jog中的速度)
	Axis_Arm[Axis_Number].Move_Relative_Velocity	:=30;	//相对运动速度
END_FOR
IF Home_Execute THEN
	Axis_Arm[1].Move_Absolute_Velocity :=10; Axis_Arm[2].Move_Absolute_Velocity :=10; Axis_Arm[3].Move_Absolute_Velocity :=10;
ELSE
	FOR Axis_Number := 1 TO 3 {BY 1} DO
			Axis_Arm[Axis_Number].Move_Absolute_Velocity	:= 10;
	END_FOR
END_IF

// =====================最大力矩规定区========================
Max_Turque_Value := 1300;

// ===============电机设置零点后到达位置规定区================
FOR Axis_Number := 1 TO 3 {BY 1} DO
	Axis_Arm[Axis_Number].Home_Absolute_Position := Model_Position[Axis_Number];
END_FOR

// ===================外部信号发生电机位置输入值================
FOR Axis_Number := 1 TO 3 {BY 1} DO
	ExSetPoint_Position[Axis_Number]:= Model_Position[Axis_Number];
END_FOR

// ===================程序与模型的变量链接===================
Robot_Simulink.stInput.t := t;								// 采样时间t与Simulink模型中的采样时间链接
//Model_Position := Robot_Simulink.stOutput.Disp_P;			// Simulink中的电机输出位移输入到控制模型
FOR Axis_Number := 1 TO 3 {BY 1} DO
	Filter_Current.stInput.Current_Motor[Axis_Number-1] := Current_Turque_Value[Axis_Number];
END_FOR	
//Current_Turque_Filter := Filter_Current.stOutput.Current_Monitor;
END_ACTION

END_PROGRAM

// ---- POUs/Welding_Robot.TcPOU
PROGRAM Welding_Robot
VAR
END_VAR

// =======================逻辑控制==========================
Robot_Simulink.stInput.t := t;											// 采样时间t与Simulink模型中的采样时间链接
//Hexapod_Robot.Model_Position := Robot_Simulink.stOutput.Disp_P;			// Simulink中的电机输出位移输入到控制模型
//Welding_Arm.Model_Position := Robot_Simulink.stOutput.Disp_P;			// Simulink中的电机输出位移输入到控制模型

END_PROGRAM

// ---- DUTs/Robot_Simulink/FB_Welding_Control_Circle_86s.TcPOU
{attribute 'TcDependOnClassFactory' := 'Welding_Control_Circle_86s'}
FUNCTION_BLOCK FB_Welding_Control_Circle_86s EXTENDS FB_TcMatSimObject
VAR_INPUT
	stInput: ST_Welding_Control_Circle_86s_Input;
END_VAR
VAR_OUTPUT
	stOutput: ST_Welding_Control_Circle_86s_Output;
END_VAR
VAR
	stInitData: ST_Welding_Control_Circle_86s_InitData;
	arrDataAreas: ARRAY[1..2] OF ST_TcMatSimObjectDataAreaInfo;
	bParametersVerified: BOOL;
END_VAR

PROPERTY CallBy_Online : TctModuleCallByType
GET
hResult := GetObjPara(16#00000000,sizeof(CallBy_Online),adr(CallBy_Online));
END_GET
SET
hResult := SetObjPara(16#00000000,sizeof(CallBy_Online),adr(CallBy_Online));
END_SET
END_PROPERTY

PROPERTY CallBy_Startup : TctModuleCallByType
GET
CallBy_Startup := stInitData.CallBy;
END_GET
SET
stInitData.CallBy := CallBy_Startup;
END_SET
END_PROPERTY

PROPERTY ContextInfoArr_0_TaskCycleTimeNs_Online : UDINT
GET
hResult := GetObjPara(16#03002080,sizeof(ContextInfoArr_0_TaskCycleTimeNs_Online),adr(ContextInfoArr_0_TaskCycleTimeNs_Online));
END_GET
SET
hResult := SetObjPara(16#03002080,sizeof(ContextInfoArr_0_TaskCycleTimeNs_Online),adr(ContextInfoArr_0_TaskCycleTimeNs_Online));
END_SET
END_PROPERTY

PROPERTY ContextInfoArr_0_TaskCycleTimeNs_Startup : UDINT
GET
ContextInfoArr_0_TaskCycleTimeNs_Startup := stInitData.ContextInfoArr_0_TaskCycleTimeNs;
END_GET
SET
stInitData.ContextInfoArr_0_TaskCycleTimeNs := ContextInfoArr_0_TaskCycleTimeNs_Startup;
END_SET
END_PROPERTY

PROPERTY ContextInfoArr_0_TaskOid_Online : OTCID
GET
hResult := GetObjPara(16#03002060,sizeof(ContextInfoArr_0_TaskOid_Online),adr(ContextInfoArr_0_TaskOid_Online));
END_GET
SET
hResult := SetObjPara(16#03002060,sizeof(ContextInfoArr_0_TaskOid_Online),adr(ContextInfoArr_0_TaskOid_Online));
END_SET
END_PROPERTY

PROPERTY ContextInfoArr_0_TaskOid_Startup : OTCID
GET
ContextInfoArr_0_TaskOid_Startup := stInitData.ContextInfoArr_0_TaskOid;
END_GET
SET
stInitData.ContextInfoArr_0_TaskOid := ContextInfoArr_0_TaskOid_Startup;
END_SET
END_PROPERTY

PROPERTY ContextInfoArr_0_TaskPort_Online : UINT
GET
hResult := GetObjPara(16#03002090,sizeof(ContextInfoArr_0_TaskPort_Online),adr(ContextInfoArr_0_TaskPort_Online));
END_GET
SET
hResult := SetObjPara(16#03002090,sizeof(ContextInfoArr_0_TaskPort_Online),adr(ContextInfoArr_0_TaskPort_Online));
END_SET
END_PROPERTY

PROPERTY ContextInfoArr_0_TaskPort_Startup : UINT
GET
ContextInfoArr_0_TaskPort_Startup := stInitData.ContextInfoArr_0_TaskPort;
END_GET
SET
stInitData.ContextInfoArr_0_TaskPort := ContextInfoArr_0_TaskPort_Startup;
END_SET
END_PROPERTY

PROPERTY ContextInfoArr_0_TaskPriority_Online : UDINT
GET
hResult := GetObjPara(16#03002070,sizeof(ContextInfoArr_0_TaskPriority_Online),adr(ContextInfoArr_0_TaskPriority_Online));
END_GET
SET
hResult := SetObjPara(16#03002070,sizeof(ContextInfoArr_0_TaskPriority_Online),adr(ContextInfoArr_0_TaskPriority_Online));
END_SET
END_PROPERTY

PROPERTY ContextInfoArr_0_TaskPriority_Startup : UDINT
GET
ContextInfoArr_0_TaskPriority_Startup := stInitData.ContextInfoArr_0_TaskPriority;
END_GET
SET
stInitData.ContextInfoArr_0_TaskPriority := ContextInfoArr_0_TaskPriority_Startup;
END_SET
END_PROPERTY

PROPERTY ContextInfoArr_0_TaskSortOrder_Online : UDINT
GET
hResult := GetObjPara(16#030020b0,sizeof(ContextInfoArr_0_TaskSortOrder_Online),adr(ContextInfoArr_0_TaskSortOrder_Online));
END_GET
SET
hResult := SetObjPara(16#030020b0,sizeof(ContextInfoArr_0_TaskSortOrder_Online),adr(ContextInfoArr_0_TaskSortOrder_Online));
END_SET
END_PROPERTY

PROPERTY ContextInfoArr_0_TaskSortOrder_Startup : UDINT
GET
ContextInfoArr_0_TaskSortOrder_Startup := stInitData.ContextInfoArr_0_TaskSortOrder;
END_GET
SET
stInitData.ContextInfoArr_0_TaskSortOrder := ContextInfoArr_0_TaskSortOrder_Startup;
END_SET
END_PROPERTY

PROPERTY CycleUpdateExecuted_Online : BOOL
GET
hResult := GetObjPara(16#00000004,sizeof(CycleUpdateExecuted_Online),adr(CycleUpdateExecuted_Online));
END_GET
SET
hResult := SetObjPara(16#00000004,sizeof(CycleUpdateExecuted_Online),adr(CycleUpdateExecuted_Online));
END_SET
END_PROPERTY

METHOD Execute : HRESULT

IF (SUCCEEDED(hResult)) THEN
  hResult := VerifyParameters();
END_IF

	// update DataArea information
SetDataAreaInfo(ADR(arrDataAreas),2);
	
	// call base method
Execute := SUPER^.Execute();
END_METHOD

PROPERTY ExecuteModelCode_Online : BOOL
GET
hResult := GetObjPara(16#00000008,sizeof(ExecuteModelCode_Online),adr(ExecuteModelCode_Online));
END_GET
SET
hResult := SetObjPara(16#00000008,sizeof(ExecuteModelCode_Online),adr(ExecuteModelCode_Online));
END_SET
END_PROPERTY

PROPERTY ExecuteModelCode_Startup : BOOL
GET
ExecuteModelCode_Startup := stInitData.ExecuteModelCode;
END_GET
SET
stInitData.ExecuteModelCode := ExecuteModelCode_Startup;
END_SET
END_PROPERTY

PROPERTY ExecutionSequence_Online : TctModuleExecutionSequenceType
GET
hResult := GetObjPara(16#00000001,sizeof(ExecutionSequence_Online),adr(ExecutionSequence_Online));
END_GET
SET
hResult := SetObjPara(16#00000001,sizeof(ExecutionSequence_Online),adr(ExecutionSequence_Online));
END_SET
END_PROPERTY

PROPERTY ExecutionSequence_Startup : TctModuleExecutionSequenceType
GET
ExecutionSequence_Startup := stInitData.ExecutionSequence;
END_GET
SET
stInitData.ExecutionSequence := ExecutionSequence_Startup;
END_SET
END_PROPERTY

METHOD FB_init : BOOL
VAR_INPUT
	/// if TRUE, the retain variables are initialized (warm start / cold start)
	bInitRetains: BOOL;
	/// if TRUE, the instance afterwards gets moved into the copy code (online change)
	bInCopyCode: BOOL;
	oid: OTCID;
END_VAR
VAR
	clsId: CLSID;
END_VAR

// initialize flags
bParametersVerified := false;
                    
// set module class id for compatibility check
clsId.Data1 := 16#4f7c9520;
clsId.Data2 := 16#5e7b;
clsId.Data3 := 16#4579;
clsId.Data4[0] := 16#be;
clsId.Data4[1] := 16#6e;
clsId.Data4[2] := 16#10;
clsId.Data4[3] := 16#c0;
clsId.Data4[4] := 16#eb;
clsId.Data4[5] := 16#37;
clsId.Data4[6] := 16#31;
clsId.Data4[7] := 16#6d;

AssignClassId(clsId);
                    
// initialize InitData structure with default values              
stInitData.CallByHdr.indexGroup := 0;
stInitData.CallByHdr.indexOffset := 16#00000000;
stInitData.CallByHdr.cbData := SIZEOF(stInitData.CallBy);
stInitData.CallBy := TctModuleCallByType.Module;
stInitData.ExecutionSequenceHdr.indexGroup := 0;
stInitData.ExecutionSequenceHdr.indexOffset := 16#00000001;
stInitData.ExecutionSequenceHdr.cbData := SIZEOF(stInitData.ExecutionSequence);
stInitData.ExecutionSequence := TctModuleExecutionSequenceType.StateUpdateAfterOutputMapping;
stInitData.StepSizeHdr.indexGroup := 0;
stInitData.StepSizeHdr.indexOffset := 16#00000002;
stInitData.StepSizeHdr.cbData := SIZEOF(stInitData.StepSize);
stInitData.StepSize := TctStepSizeType.UseTaskCycleTime;
stInitData.ExecuteModelCodeHdr.indexGroup := 0;
stInitData.ExecuteModelCodeHdr.indexOffset := 16#00000008;
stInitData.ExecuteModelCodeHdr.cbData := SIZEOF(stInitData.ExecuteModelCode);
stInitData.ExecuteModelCode := 1;
stInitData.ContextInfoArr_0_TaskOidHdr.indexGroup := 0;
stInitData.ContextInfoArr_0_TaskOidHdr.indexOffset := 16#03002060;
stInitData.ContextInfoArr_0_TaskOidHdr.cbData := SIZEOF(stInitData.ContextInfoArr_0_TaskOid);
stInitData.ContextInfoArr_0_TaskPriorityHdr.indexGroup := 0;
stInitData.ContextInfoArr_0_TaskPriorityHdr.indexOffset := 16#03002070;
stInitData.ContextInfoArr_0_TaskPriorityHdr.cbData := SIZEOF(stInitData.ContextInfoArr_0_TaskPriority);
stInitData.ContextInfoArr_0_TaskCycleTimeNsHdr.indexGroup := 0;
stInitData.ContextInfoArr_0_TaskCycleTimeNsHdr.indexOffset := 16#03002080;
stInitData.ContextInfoArr_0_TaskCycleTimeNsHdr.cbData := SIZEOF(stInitData.ContextInfoArr_0_TaskCycleTimeNs);
stInitData.ContextInfoArr_0_TaskPortHdr.indexGroup := 0;
stInitData.ContextInfoArr_0_TaskPortHdr.indexOffset := 16#03002090;
stInitData.ContextInfoArr_0_TaskPortHdr.cbData := SIZEOF(stInitData.ContextInfoArr_0_TaskPort);
stInitData.ContextInfoArr_0_TaskSortOrderHdr.indexGroup := 0;
stInitData.ContextInfoArr_0_TaskSortOrderHdr.indexOffset := 16#030020b0;
stInitData.ContextInfoArr_0_TaskSortOrderHdr.cbData := SIZEOF(stInitData.ContextInfoArr_0_TaskSortOrder);
stInitData.Header.cbData := SIZEOF(stInitData)-SIZEOF(stInitData.Header);
stInitData.Header.uiElmCnt := 9;


// set pointer to InitData structure
SetInitDataInfo(ADR(stInitData));

// set DataArea information
SetDataAreaInfo(ADR(arrDataAreas),2);
arrDataAreas[1].nDataAreaId := 0;
arrDataAreas[1].nSize := SIZEOF(stInput);
arrDataAreas[1].pPlcVar := ADR(stInput);
arrDataAreas[1].pModuleProcImg := 0;
arrDataAreas[1].eDataAreaType := E_TcMatSimDataAreaType.InputDst;
arrDataAreas[2].nDataAreaId := 1;
arrDataAreas[2].nSize := SIZEOF(stOutput);
arrDataAreas[2].pPlcVar := ADR(stOutput);
arrDataAreas[2].pModuleProcImg := 0;
arrDataAreas[2].eDataAreaType := E_TcMatSimDataAreaType.OutputSrc;


// initialize basic interface pointers and return
FB_init := SUCCEEDED(Init(oid));
END_METHOD

PROPERTY InitData : ST_Welding_Control_Circle_86s_InitData
GET
InitData := stInitData;
END_GET
SET
stInitData := InitData;
END_SET
END_PROPERTY

PROPERTY Input_Online : ExtU_output_WeldingDiameter10_T
GET
hResult := GetObjPara(16#80000000,sizeof(Input_Online),adr(Input_Online));
END_GET
SET
hResult := SetObjPara(16#80000000,sizeof(Input_Online),adr(Input_Online));
END_SET
END_PROPERTY

{attribute 'object_name' := 'Internal_SetObjState'}
METHOD PROTECTED Internal_SetObjState
VAR_INPUT
	hr: REFERENCE TO HRESULT;
	nextState: TCOM_STATE;
END_VAR

// update pointer to InitData structure
SetInitDataInfo(ADR(stInitData));
// call base method
SUPER^.Internal_SetObjState(hr,nextState);
END_METHOD

PROPERTY MdlInitialized_Online : BOOL
GET
hResult := GetObjPara(16#00000003,sizeof(MdlInitialized_Online),adr(MdlInitialized_Online));
END_GET
SET
hResult := SetObjPara(16#00000003,sizeof(MdlInitialized_Online),adr(MdlInitialized_Online));
END_SET
END_PROPERTY

PROPERTY ModuleBuildInfo_Online : TctModuleBuildInfoType
GET
hResult := GetObjPara(16#00000007,sizeof(ModuleBuildInfo_Online),adr(ModuleBuildInfo_Online));
END_GET
SET
hResult := SetObjPara(16#00000007,sizeof(ModuleBuildInfo_Online),adr(ModuleBuildInfo_Online));
END_SET
END_PROPERTY

PROPERTY ModuleInfo_Online : TctModuleInfoType
GET
hResult := GetObjPara(16#00000006,sizeof(ModuleInfo_Online),adr(ModuleInfo_Online));
END_GET
SET
hResult := SetObjPara(16#00000006,sizeof(ModuleInfo_Online),adr(ModuleInfo_Online));
END_SET
END_PROPERTY

{attribute 'object_name' := 'SaveOnlineParametersForInit'}
METHOD SaveOnlineParametersForInit : HRESULT
VAR
	idx: UINT;
	pInitElemHdr: POINTER TO TComInitDataElmHdr;
	pData: PVOID;
	nData: UDINT;
END_VAR
VAR CONSTANT
	nInitDataAlignment: UDINT := 4;
END_VAR

// update pointer to InitData structure
SetInitDataInfo(ADR(stInitData));
// call base method
SaveOnlineParametersForInit := SUPER^.SaveOnlineParametersForInit();
END_METHOD

PROPERTY SimulinkTime_Online : LREAL
GET
hResult := GetObjPara(16#00000005,sizeof(SimulinkTime_Online),adr(SimulinkTime_Online));
END_GET
SET
hResult := SetObjPara(16#00000005,sizeof(SimulinkTime_Online),adr(SimulinkTime_Online));
END_SET
END_PROPERTY

PROPERTY StepSize_Online : TctStepSizeType
GET
hResult := GetObjPara(16#00000002,sizeof(StepSize_Online),adr(StepSize_Online));
END_GET
SET
hResult := SetObjPara(16#00000002,sizeof(StepSize_Online),adr(StepSize_Online));
END_SET
END_PROPERTY

PROPERTY StepSize_Startup : TctStepSizeType
GET
StepSize_Startup := stInitData.StepSize;
END_GET
SET
stInitData.StepSize := StepSize_Startup;
END_SET
END_PROPERTY

{attribute 'object_name' := 'VerifyParameters'}
METHOD PRIVATE VerifyParameters : HRESULT
VAR
	moduleCallByParam: TctModuleCallByType;
END_VAR

IF (bParametersVerified) THEN
  VerifyParameters := Tc2_System.E_HRESULTAdsErr.HRESULT_ADS_NOERROR;
ELSE
  VerifyParameters := GetObjPara(stInitData.CallByHdr.indexOffset,SIZEOF(moduleCallByParam),ADR(moduleCallByParam));
  
  // check the "CallBy" parameter to be set to "Module"
  IF (SUCCEEDED(VerifyParameters) AND (moduleCallByParam <> TctModuleCallByType.Module)) THEN
      VerifyParameters := Tc2_System.E_HRESULTAdsErr.INVALIDPARM;
  END_IF
  
  // set the parameters verified flag
  bParametersVerified := SUCCEEDED(VerifyParameters);
END_IF
END_METHOD

END_FUNCTION_BLOCK

// ---- DUTs/Robot_Simulink/FB_TcMatSimObject.TcPOU
FUNCTION_BLOCK FB_TcMatSimObject
VAR_INPUT
	/// set this flag to write FB input values to the TcComObject's input DataAreas. This will overwrite the mapped input values before module execution. Set to FALSE to read the mapped input values from the TcComObject to the FB.
	bWriteFbInputValues: BOOL := TRUE;
END_VAR
VAR
	/// process image src and dst pointers and sizes
	pDataAreas: POINTER TO ST_TcMatSimObjectDataAreaInfo;
	nDataAreas: UDINT;
	/// global interface pointers
	ipObjSrv: ITComObjectServer;
	/// object interface pointers
	ipTcComObj: ITComObject;
	ipTcCyclic: ITcCyclic;
	ipTcPostCyclic: ITcPostCyclic;
	ipTcAdi: ITcADI;
	/// task interface pointers
	ipTask: ITcTask;
	/// initial parameters
	pInitData: POINTER TO TComInitDataHdr;
	/// hResult of interface calls (0 if no error)
	hResult: HRESULT;
	/// module class ID
	moduleClsId: CLSID;
	/// expected/desired module class ID
	assignedClsId: CLSID;
	bClassIdVerified: BOOL;
	/// flag indicating whether the module instance was created dynamically
	bDynInstance: BOOL;
	/// the object state at the time FB_init was called, FB_exit will try to switch to this state (only if this means to shift down)
	eInitialObjState: TCOM_STATE := TCOM_STATE.TCOM_STATE_INIT;
END_VAR

METHOD PUBLIC AssignClassId
VAR_INPUT
	clsId : CLSID;
END_VAR
assignedClsId := clsId;
bClassIdVerified := false;
END_METHOD

PROPERTY ClassId : CLSID
GET
hResult := ReadModuleClassId();
ClassId := moduleClsId;
END_GET
END_PROPERTY

PROPERTY Error : BOOL
GET
Error := FAILED(hResult);
END_GET
END_PROPERTY

PROPERTY ErrorCode : HRESULT
GET
ErrorCode := hResult;
END_GET
END_PROPERTY

{attribute 'object_name' := 'Execute'}
METHOD Execute : HRESULT
VAR
	nDaIdx: UDINT;
	pCurDataArea: POINTER TO ST_TcMatSimObjectDataAreaInfo;
END_VAR

IF (SUCCEEDED(hResult)) THEN
  hResult := VerifyClassId();
END_IF

IF (SUCCEEDED(hResult) AND State<>TCOM_STATE_OP) THEN
  hResult := Tc2_System.E_HRESULTAdsErr.NOTREADY;
END_IF

// get image pointers
IF (SUCCEEDED(hResult)) THEN
  GetImagePtrs(hResult);
END_IF

// copy inputs
IF (pDataAreas<>0 AND bWriteFbInputValues) THEN
  FOR nDaIdx:=0 TO nDataAreas-1 DO
    IF (FAILED(hResult))THEN
      CONTINUE;
    END_IF
    pCurDataArea := pDataAreas + nDaIdx*SIZEOF(ST_TcMatSimObjectDataAreaInfo);
    IF ((pCurDataArea^.eDataAreaType <> E_TcMatSimDataAreaType.InputDst))THEN
      CONTINUE;
    END_IF
    IF (pCurDataArea^.pModuleProcImg<>0 AND pCurDataArea^.pPlcVar<>0) THEN
      MEMCPY(pCurDataArea^.pModuleProcImg,pCurDataArea^.pPlcVar,pCurDataArea^.nSize);
    ELSE
      hResult := Tc2_System.E_HRESULTAdsErr.NOINTERFACE;
    END_IF
  END_FOR
END_IF

// call cycle update
IF (SUCCEEDED(hResult)) THEN
  IF (ipTcCyclic<>0) THEN
    hResult := ipTcCyclic.CycleUpdate(ipTask:= ipTask, ipCaller:= 0, context:= 0);
  ELSE
    hResult := Tc2_System.E_HRESULTAdsErr.NOINTERFACE;
  END_IF
END_IF

// copy outputs
IF (pDataAreas<>0) THEN
  FOR nDaIdx:=0 TO nDataAreas-1 DO
    IF (FAILED(hResult))THEN
      CONTINUE;
    END_IF
    pCurDataArea := pDataAreas + nDaIdx*SIZEOF(ST_TcMatSimObjectDataAreaInfo);
    IF ((pCurDataArea^.eDataAreaType = E_TcMatSimDataAreaType.OutputSrc) OR NOT bWriteFbInputValues) THEN
      IF (pCurDataArea^.pModuleProcImg<>0 AND pCurDataArea^.pPlcVar<>0) THEN
        MEMCPY(pCurDataArea^.pPlcVar,pCurDataArea^.pModuleProcImg,pCurDataArea^.nSize);
      ELSE
        hResult := Tc2_System.E_HRESULTAdsErr.NOINTERFACE;
      END_IF
    END_IF
  END_FOR
END_IF


// call post cyclic update
IF (SUCCEEDED(hResult)) THEN
  IF (ipTcPostCyclic<>0) THEN
    hResult := ipTcPostCyclic.PostCyclicUpdate(ipTask:= 0, ipCaller:= 0, context:= 0);
  ELSE
    hResult := Tc2_System.E_HRESULTAdsErr.NOINTERFACE;
  END_IF
END_IF

ReleaseImagePtrs();

Execute := hResult;
END_METHOD

{attribute 'object_name' := 'FB_exit'}
METHOD FB_exit : BOOL
VAR_INPUT
	/// Online Change
	bInCopyCode: BOOL;
END_VAR

IF (NOT bInCopyCode) THEN
  IF (ipObjSrv<>0) THEN
    ipObjSrv.TcRelease();
    ipObjSrv := 0;
  END_IF

  ReleaseTcComInterface();
END_IF
END_METHOD

{attribute 'object_name' := 'FB_init'}
METHOD FB_init : BOOL
VAR_INPUT
	/// init retain variables
	bInitRetains: BOOL;
	/// Online Change
	bInCopyCode: BOOL;
	oid: OTCID;
END_VAR

FB_init := SUCCEEDED(Init(oid));
END_METHOD

{attribute 'object_name' := 'GetImagePtrs'}
METHOD PRIVATE GetImagePtrs
VAR_INPUT
	hr: REFERENCE TO HRESULT;
END_VAR
VAR
	nDaIdx: UDINT;
	pCurDataArea: POINTER TO ST_TcMatSimObjectDataAreaInfo;
END_VAR

IF (ipTcAdi=0) THEN
  hr := Tc2_System.E_HRESULTAdsErr.NOINTERFACE;
END_IF
IF(State<>TCOM_STATE_OP)THEN
  hr := Tc2_System.E_HRESULTAdsErr.INVALIDSTATE;
END_IF


// get pointers to process images
IF (pDataAreas<>0) THEN
  FOR nDaIdx:=0 TO nDataAreas-1 DO
    pCurDataArea := pDataAreas + nDaIdx*SIZEOF(ST_TcMatSimObjectDataAreaInfo);
    IF (FAILED(hr))THEN
      CONTINUE;
    END_IF
    IF ((pCurDataArea^.eDataAreaType <> E_TcMatSimDataAreaType.InputDst) AND (pCurDataArea^.eDataAreaType <> E_TcMatSimDataAreaType.OutputSrc))THEN
      CONTINUE;
    END_IF
    IF (pCurDataArea^.pModuleProcImg=0 AND pCurDataArea^.nSize>0) THEN
      hr := ipTcAdi.GetImagePtr(size:= pCurDataArea^.nSize , offs:=0 , adi_x:=pCurDataArea^.nDataAreaId , ppData:=ADR(pCurDataArea^.pModuleProcImg));
    END_IF
  END_FOR
END_IF

IF (FAILED(hr)) THEN
  ReleaseImagePtrs();
END_IF
END_METHOD

{attribute 'object_name' := 'GetObjPara'}
METHOD GetObjPara : HRESULT
VAR_INPUT
	pid: PTCID;
	nData: UDINT;
	pData: PVOID;
END_VAR

IF (ipTcComObj=0) THEN
  GetObjPara := Tc2_System.E_HRESULTAdsErr.NOINTERFACE;
END_IF

IF (SUCCEEDED(GetObjPara)) THEN
  GetObjPara := ipTcComObj.TcGetObjPara(pid:=pid,nData,pData,0);
END_IF
END_METHOD

{attribute 'object_name' := 'Init'}
METHOD PROTECTED Init : HRESULT
VAR_INPUT
	oid: OTCID;
END_VAR

// preinitialize variables
memset(ADR(moduleClsId),0,SIZEOF(moduleClsId));
bClassIdVerified := FALSE;
hResult := Tc2_System.E_HRESULTAdsErr.HRESULT_ADS_NOERROR;

// get object server
IF (ipObjSrv=0) THEN
  hResult := FW_ObjMgr_GetObjectServer(_AppInfo.ObjId,ADR(ipObjSrv));
END_IF

// try to get object interfaces
IF (SUCCEEDED(hresult)) THEN
  QueryTcComInterface(hResult,oid);
END_IF

// verify class id
IF (SUCCEEDED(hresult)) THEN
  hresult := VerifyClassId();
END_IF

// query interfaces, if the current state is higher than INIT
IF (SUCCEEDED(hresult) AND State>TCOM_STATE.TCOM_STATE_INIT) THEN
  QueryObjInterfaces(hResult);
END_IF

// return value
Init := hresult;
END_METHOD

{attribute 'object_name' := 'InitObjName'}
METHOD PRIVATE InitObjName
VAR_INPUT
	hr: REFERENCE TO HRESULT;
END_VAR
VAR
	objectName: STRING(255) := 'TempContr_PlcRtFbInstance';
	oid: OTCID;
END_VAR

IF (SUCCEEDED(hr)) THEN
  hr := ipTcComObj.TcGetObjectId(oid);
END_IF

IF (SUCCEEDED(hr) and bDynInstance) THEN
  objectName := TC2_STANDARD.CONCAT(objectName,'_');
  objectName := TC2_STANDARD.CONCAT(objectName,UDINT_TO_STRING(oid));
  hr := ipTcComObj.TcSetObjectName(ADR(objectName));
END_IF
END_METHOD

{attribute 'object_name' := 'Internal_SetObjState'}
METHOD PROTECTED Internal_SetObjState
VAR_INPUT
	hr: REFERENCE TO HRESULT;
	nextState: TCOM_STATE;
END_VAR

// verify class id
IF (SUCCEEDED(hr)) THEN
  hr := VerifyClassId();
END_IF

// switch object state
IF (SUCCEEDED(hr) AND nextState>=TCOM_STATE_INIT) THEN
  IF (ipTcComObj=0) THEN
    hr := Tc2_System.E_HRESULTAdsErr.NOINTERFACE;
  END_IF
  IF (ipObjSrv=0) THEN
    hr := Tc2_System.E_HRESULTAdsErr.NOINTERFACE;
  END_IF
  IF (SUCCEEDED(hr)) THEN
    hr := ipTcComObj.TcSetObjState(nextState,ipObjSrv,pInitData);
  END_IF
END_IF
END_METHOD

{attribute 'object_name' := 'QueryObjInterface'}
METHOD PRIVATE QueryObjInterface
VAR_INPUT
	hr: REFERENCE TO HRESULT;
	iid: REFERENCE TO IID;
	pipItf: POINTER TO ITcUnknown;
END_VAR
VAR CONSTANT
	pNull: PVOID := 0;
END_VAR

IF (SUCCEEDED(hr)) THEN
  IF (ipTcComObj=0) THEN
    hr := Tc2_System.E_HRESULTAdsErr.NOINTERFACE;
  ELSIF (pipItf^=ULINT_TO_DWORD(pNull)) THEN
    hr := ipTcComObj.TcQueryInterface(iid:= iid, pipItf:=pipItf);
  END_IF
END_IF
END_METHOD

{attribute 'object_name' := 'QueryObjInterfaces'}
METHOD PRIVATE QueryObjInterfaces
VAR_INPUT
	hr: REFERENCE TO HRESULT;
END_VAR

IF(State<TCOM_STATE_PREOP)THEN
  hr := Tc2_System.E_HRESULTAdsErr.INVALIDSTATE;
END_IF

//cyclic interface
QueryObjInterface(hr,IID_ITCCYCLIC,ADR(ipTcCyclic));
//post cyclic interface
QueryObjInterface(hr,IID_ITCPOSTCYCLIC,ADR(ipTcPostCyclic));
//adi interface
QueryObjInterface(hr,IID_ITcADI,ADR(ipTcAdi));
END_METHOD

{attribute 'object_name' := 'QueryTcComInterface'}
METHOD PRIVATE QueryTcComInterface
VAR_INPUT
	hr: REFERENCE TO HRESULT;
	oid: OTCID;
END_VAR

IF (ipObjSrv=0) THEN
  hr := Tc2_System.E_HRESULTAdsErr.NOINTERFACE;
END_IF

IF (SUCCEEDED(hr) AND ipTcComObj=0) THEN
  bDynInstance := FALSE;
  IF(oid>0) THEN
    // query interface of existing object
    hr := ipObjSrv.TcQueryObjectInterface(oid,IID_ITComObject,ADR(ipTcComObj));
  ELSE
    // create new instance and get the object interface
    hr := ipObjSrv.TcCreateInstance(assignedClsId,IID_ITComObject,ADR(ipTcComObj));
    IF (SUCCEEDED(hr)) THEN
      bDynInstance := TRUE;
      hr := ipTcComObj.TcSetObjectId(OTCID_CreateNewId);
    END_IF
  END_IF
  IF (SUCCEEDED(hr)) THEN
    eInitialObjState := State;
  END_IF
END_IF
END_METHOD

{attribute 'object_name' := 'ReadModuleClassId'}
METHOD PRIVATE ReadModuleClassId : HRESULT
VAR
	emptyClsId: CLSID;
END_VAR
memset(ADR(emptyClsId),0,SIZEOF(emptyClsId));
IF (memcmp(ADR(moduleClsId),ADR(emptyClsId),SIZEOF(moduleClsId))=0) THEN
  IF (ipTcComObj=0) THEN
    ReadModuleClassId := Tc2_System.E_HRESULTAdsErr.NOINTERFACE;
  END_IF

  //objectClsId := clsid;
  IF (SUCCEEDED(ReadModuleClassId)) THEN
    ReadModuleClassId := ipTcComObj.GetClassId(moduleClsId);
  END_IF
END_IF
END_METHOD

{attribute 'object_name' := 'ReleaseImagePtrs'}
METHOD PRIVATE ReleaseImagePtrs : HRESULT
VAR
	nDaIdx: UDINT;
	pCurDataArea: POINTER TO ST_TcMatSimObjectDataAreaInfo;
END_VAR

IF (ipTcAdi=0) THEN
  ReleaseImagePtrs := Tc2_System.E_HRESULTAdsErr.NOINTERFACE;
END_IF

IF (SUCCEEDED(ReleaseImagePtrs) AND pDataAreas<>0) THEN
  // release pointers to the simulink module process images
  FOR nDaIdx:=0 TO nDataAreas-1 DO
    pCurDataArea := pDataAreas + nDaIdx*SIZEOF(ST_TcMatSimObjectDataAreaInfo);

    IF (pCurDataArea^.pModuleProcImg<>0) THEN
      ipTcAdi.ReleaseImagePtr(pData:=pCurDataArea^.pModuleProcImg);
      pCurDataArea^.pModuleProcImg := 0;
    END_IF
  END_FOR
END_IF
END_METHOD

{attribute 'object_name' := 'ReleaseObjInterfaces'}
METHOD PRIVATE ReleaseObjInterfaces : HRESULT

// release interface pointers
IF (ipTcCyclic<>0) THEN
  ipTcCyclic.TcRelease();
  ipTcCyclic := 0;
END_IF
IF (ipTcPostCyclic<>0) THEN
  ipTcPostCyclic.TcRelease();
  ipTcPostCyclic := 0;
END_IF
IF (ipTcAdi<>0) THEN
  ipTcAdi.TcRelease();
  ipTcAdi := 0;
END_IF
END_METHOD

{attribute 'object_name' := 'ReleaseTcComInterface'}
METHOD PRIVATE ReleaseTcComInterface : HRESULT
VAR
	nStateChangeCnt: DINT := 0;
END_VAR

IF (ipTcComObj<>0) THEN
  WHILE (State>eInitialObjState AND nStateChangeCnt<1000) DO
    State := eInitialObjState;
    nStateChangeCnt := nStateChangeCnt+1;
  END_WHILE
  ReleaseObjInterfaces();
  IF (bDynInstance) THEN
    ReleaseTcComInterface := TC3_MODULE.FW_ObjMgr_DeleteInstance(ADR(ipTcComObj));
  ELSE
    ipTcComObj.TcRelease();
  END_IF
  ipTcComObj := 0;
END_IF
END_METHOD

{attribute 'object_name' := 'ResetHresult'}
METHOD ResetHresult
hResult := S_OK;
END_METHOD

{attribute 'object_name' := 'SaveOnlineParametersForInit'}
METHOD SaveOnlineParametersForInit : HRESULT
VAR
	idx: UINT;
	pInitElemHdr: POINTER TO TComInitDataElmHdr;
	pData: PVOID;
	nData: UDINT;
END_VAR
VAR CONSTANT
	nInitDataAlignment: UDINT := 4;
END_VAR
IF (pInitData<>0) THEN
  pInitElemHdr := pInitData + SIZEOF(pInitData^);
  FOR idx:=1 TO pInitData^.uiElmCnt DO
    pData := pInitElemHdr + ULINT_TO_DWORD(SIZEOF(pInitElemHdr^));
    nData := pInitElemHdr^.cbData;
    SaveOnlineParametersForInit := GetObjPara(pInitElemHdr^.indexOffset,nData,pData);
    IF (FAILED(SaveOnlineParametersForInit)) THEN
      RETURN;
    END_IF
    pInitElemHdr := pData + (nInitDataAlignment*((nData + nInitDataAlignment - 1)/nInitDataAlignment));
  END_FOR
ELSE
	SaveOnlineParametersForInit := Tc2_System.E_HRESULTAdsErr.NOTINIT;
END_IF
END_METHOD


METHOD PUBLIC SetDataAreaInfo
VAR_INPUT
  pDataAreas: POINTER TO ST_TcMatSimObjectDataAreaInfo;
  nDataAreas: UDINT;
END_VAR

THIS^.nDataAreas := nDataAreas;
THIS^.pDataAreas := pDataAreas;
END_METHOD


METHOD PUBLIC SetInitDataInfo
VAR_INPUT
  pInitData : POINTER TO TComInitDataHdr;
END_VAR
this^.pInitData := pInitData;
END_METHOD

{attribute 'object_name' := 'SetObjPara'}
METHOD SetObjPara : HRESULT
VAR_INPUT
	pid: PTCID;
	nData: UDINT;
	pData: PVOID;
END_VAR

IF (ipTcComObj=0) THEN
  SetObjPara := Tc2_System.E_HRESULTAdsErr.NOINTERFACE;
END_IF

IF (SUCCEEDED(SetObjPara)) THEN
  SetObjPara := ipTcComObj.TcSetObjPara(pid:=pid,nData,pData,0);
END_IF
END_METHOD

{attribute 'object_name' := 'SetObjState'}
METHOD SetObjState : HRESULT
VAR_INPUT
	finalState: TCOM_STATE;
END_VAR
VAR
	bShiftUp: BOOL;
	bShiftDown: BOOL;
	currentState: TCOM_STATE;
END_VAR

currentState := State;

bShiftUp := finalState>currentState;
bShiftDown := finalState<currentState;

// do not switch up on error
IF (FAILED(hresult)) THEN
  bShiftUp := FALSE;
END_IF
// reset existing error on switching down
IF (bShiftDown) THEN
  ResetHresult();
END_IF

// prepared state switch
CASE currentState OF
  TCOM_STATE_INIT:
    IF(bShiftUp) THEN
      QueryTcComInterface(hResult,0);
      Internal_SetObjState(hResult,TCOM_STATE.TCOM_STATE_PREOP);
      InitObjName(hResult);
    END_IF

  TCOM_STATE_PREOP:
    IF(bShiftUp) THEN
      Internal_SetObjState(hResult,TCOM_STATE.TCOM_STATE_SAFEOP);
      QueryObjInterfaces(hResult);
    ELSIF (bShiftDown) THEN
      Internal_SetObjState(hResult,TCOM_STATE.TCOM_STATE_INIT);
    END_IF

  TCOM_STATE_SAFEOP:
    IF(bShiftUp) THEN
      Internal_SetObjState(hResult,TCOM_STATE.TCOM_STATE_OP);
      QueryObjInterfaces(hResult);
    ELSIF (bShiftDown) THEN
      Internal_SetObjState(hResult,TCOM_STATE.TCOM_STATE_PREOP);
      ReleaseObjInterfaces();
    END_IF


  TCOM_STATE_OP:
    IF (bShiftDown) THEN
      Internal_SetObjState(hResult,TCOM_STATE.TCOM_STATE_SAFEOP);
    END_IF
END_CASE

SetObjState := hResult;
END_METHOD

PROPERTY State : TCOM_STATE
GET
VAR
	hr: HRESULT := S_OK;
	eObjState: TCOM_STATE;
END_VAR

IF (ipTcComObj<>0) THEN
  hr := ipTcComObj.TcGetObjState(ADR(eObjState));
IF (FAILED(hr)) THEN
  eObjState := TCOM_STATE.TCOM_STATE_INIT;
END_IF
ELSE
  eObjState := TCOM_STATE.TCOM_STATE_INIT;
END_IF
State := eObjState;
END_GET
SET
SetObjState(State);
END_SET
END_PROPERTY

{attribute 'object_name' := 'VerifyClassId'}
METHOD PRIVATE VerifyClassId : HRESULT
VAR
	emptyClsId: CLSID;
END_VAR
memset(ADR(emptyClsId),0,SIZEOF(emptyClsId));
IF (bClassIdVerified) THEN
  // class ID was already verified
  VerifyClassId := Tc2_System.E_HRESULTAdsErr.HRESULT_ADS_NOERROR;
ELSIF (memcmp(ADR(assignedClsId),ADR(emptyClsId),SIZEOF(assignedClsId))=0) THEN
  // skip class ID verification if no assignedClsId specified
  VerifyClassId := Tc2_System.E_HRESULTAdsErr.HRESULT_ADS_NOERROR;
ELSE
  // verify class ID
  VerifyClassId := ReadModuleClassId();

  IF (SUCCEEDED(VerifyClassId)) THEN
    IF (memcmp(ADR(assignedClsId),ADR(moduleClsId),SIZEOF(assignedClsId))<>0) THEN
     VerifyClassId := Tc2_System.E_HRESULTAdsErr.INVALIDCLSID;
    END_IF
  END_IF
  bClassIdVerified := SUCCEEDED(VerifyClassId);
END_IF
END_METHOD

END_FUNCTION_BLOCK

// ---- GlobalTextList.TcGTLO
TEXTLIST GlobalTextList
  145 = ' %.2f'
  165 = ' t_Interval=%.2f'
  167 = ' t_Interval=%.3f'
  169 = ' t_Interval=%.4f'
  168 = ' t_Interval=%.5f'
  143 = '%.2f'
  81 = 'Axis10_Back'
  82 = 'Axis10_Home'
  117 = 'Axis10_Move'
  11 = 'Axis10_Power'
  83 = 'Axis11_Back'
  84 = 'Axis11_Home'
  118 = 'Axis11_Move'
  12 = 'Axis11_Power'
  85 = 'Axis12_Back'
  86 = 'Axis12_Home'
  119 = 'Axis12_Move'
  13 = 'Axis12_Power'
  87 = 'Axis13_Back'
  88 = 'Axis13_Home'
  120 = 'Axis13_Move'
  14 = 'Axis13_Power'
  89 = 'Axis14_Back'
  90 = 'Axis14_Home'
  121 = 'Axis14_Move'
  15 = 'Axis14_Power'
  91 = 'Axis15_Back'
  92 = 'Axis15_Home'
  122 = 'Axis15_Move'
  16 = 'Axis15_Power'
  93 = 'Axis16_Back'
  94 = 'Axis16_Home'
  123 = 'Axis16_Move'
  17 = 'Axis16_Power'
  95 = 'Axis17_Back'
  96 = 'Axis17_Home'
  124 = 'Axis17_Move'
  18 = 'Axis17_Power'
  97 = 'Axis18_Back'
  98 = 'Axis18_Home'
  125 = 'Axis18_Move'
  19 = 'Axis18_Power'
  62 = 'Axis1_Back'
  64 = 'Axis1_Home'
  63 = 'Axis1_Home_Set'
  106 = 'Axis1_M'
  108 = 'Axis1_Move'
  2 = 'Axis1_Power'
  65 = 'Axis2_Back'
  66 = 'Axis2_Home'
  109 = 'Axis2_Move'
  3 = 'Axis2_Power'
  67 = 'Axis3_Back'
  68 = 'Axis3_Home'
  110 = 'Axis3_Move'
  4 = 'Axis3_Power'
  69 = 'Axis4_Back'
  70 = 'Axis4_Home'
  111 = 'Axis4_Move'
  5 = 'Axis4_Power'
  71 = 'Axis5_Back'
  72 = 'Axis5_Home'
  112 = 'Axis5_Move'
  6 = 'Axis5_Power'
  73 = 'Axis6_Back'
  74 = 'Axis6_Home'
  113 = 'Axis6_Move'
  7 = 'Axis6_Power'
  75 = 'Axis7_Back'
  76 = 'Axis7_Home'
  114 = 'Axis7_Move'
  8 = 'Axis7_Power'
  77 = 'Axis8_Back'
  78 = 'Axis8_Home'
  115 = 'Axis8_Move'
  9 = 'Axis8_Power'
  79 = 'Axis9_Back'
  80 = 'Axis9_Home'
  116 = 'Axis9_Move'
  10 = 'Axis9_Power'
  56 = 'Axis_ActPostion[INDEX]'
  171 = 'Axis_ActPostion[Robot]'
  60 = 'Back'
  57 = 'Current_Turque_Value[INDEX]'
  172 = 'Current_Turque_Value[Robot]'
  39 = 'Driver10_Reset'
  40 = 'Driver11_Reset'
  41 = 'Driver12_Reset'
  42 = 'Driver13_Reset'
  43 = 'Driver14_Reset'
  44 = 'Driver15_Reset'
  45 = 'Driver16_Reset'
  46 = 'Driver17_Reset'
  47 = 'Driver18_Reset'
  30 = 'Driver1_Reset'
  31 = 'Driver2_Reset'
  32 = 'Driver3_Reset'
  33 = 'Driver4_Reset'
  34 = 'Driver5_Reset'
  35 = 'Driver6_Reset'
  36 = 'Driver7_Reset'
  37 = 'Driver8_Reset'
  38 = 'Driver9_Reset'
  127 = 'Error & Reset'
  126 = 'Error&Reset'
  151 = 'Exsetopint_Enable'
  152 = 'Exsetopint_On'
  141 = 'Exsetpoint_Exectue'
  23 = 'Home'
  59 = 'Home_Execute'
  61 = 'Home_Set'
  131 = 'Leg1_Home'
  132 = 'Leg2_Home'
  133 = 'Leg3_Home'
  134 = 'Leg4_Home'
  135 = 'Leg5_Home'
  136 = 'Leg6_Home'
  130 = 'Move & Stand'
  107 = 'MoveAbsoluteDone[INDEX]'
  129 = 'Move_Execute'
  53 = 'Power'
  20 = 'Power_Execute'
  29 = 'Reset'
  49 = 'Reset_Execute'
  26 = 'Robot_Error'
  101 = 'Robot_Home_Set'
  0 = 'Robot_Power'
  48 = 'Robot_Reset'
  128 = 'Robot_Stand_Execute'
  99 = 'Robot_Start_Back'
  100 = 'sadad'
  166 = 'Simulink_Move'
  147 = 't=%.2f'
  170 = 't=%.3f'
  144 = 'T_ALL = %.2f'
  158 = 't_Interval=%.2f'
  22 = '切换视图'
  157 = '取样时间间隔 t_Interval'
  160 = '取样时间间隔 t_Interval(ms)'
  161 = '取样时间间隔 t_Interval(s)'
  159 = '取样时间间隔 t_Interval/ms'
  139 = '可以用来整体机器人运动'
  140 = '可以用来整体机器人进行Simulink模型验证'
  104 = '可以用来给单个四缸伸长或者是整体机器人站立'
  28 = '可以用来给单个电机或者是整体机器人上电'
  55 = '可以用来给单个电机或者是整体机器人找零'
  103 = '可以用来给单个电机或者是整体机器人站立'
  52 = '可以用来错误时给单个电机或者是整体机器人进行驱动重置'
  24 = '否'
  149 = '开始输入轨迹'
  156 = '当前取样时间 t'
  163 = '当前取样时间 t(s)'
  25 = '是'
  148 = '是否开始输入轨迹'
  21 = '是否进行上电操作'
  58 = '是否进行找零操作'
  1 = '是否进行整机操作'
  142 = '是否进行运动操作'
  50 = '是否进行驱动重置'
  138 = '本界面为电机Sumulink模型运动程序：'
  137 = '本界面为电机Sumulink程序：'
  27 = '本界面为电机上电程序：'
  102 = '本界面为电机伸长/机器人站立程序：'
  54 = '本界面为电机找零程序：'
  105 = '本界面为电机绝对运动/机器人站立程序：'
  51 = '本界面为驱动重置程序：'
  154 = '输入运动总时长 T_ALL'
  162 = '输入运动总时长 T_ALL(s)'
  150 = '运动当前时间 t'
  164 = '运动当前时间 t(s)'
  146 = '运动总时长 T_ALL'
  155 = '运动时间间隔 t'
  153 = '运动终止信号'
END_TEXTLIST

// ---- VISUs/Visu_Home.TcVIS
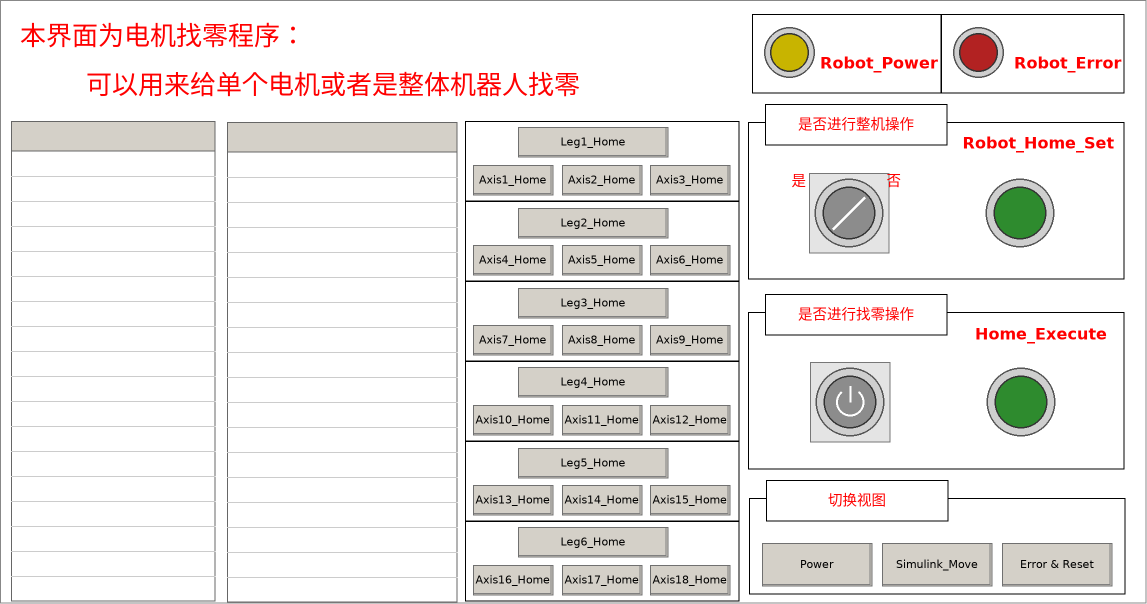
VISUALIZATION Visu_Home  // 1147x604
    Rectangle (752,14 189x79)
    Rectangle (748,312 376x157)
    Label (964,318 154x32), "Home_Execute"
    Rectangle (765,294 182x41), "是否进行找零操作"
    Lamp1 (981,362 80x80), variable: Home_Execute, style: Lamp-Lamp1-Green
    PowerSwitch (810,362 80x80), variable: Home_Execute, behaviour: TOGGLE, style: Switch-PowerSwitch-Gray
    Rectangle (941,14 183x79)
    Lamp1 (948,23 61x59), variable: Hexapod_Robot.Robot_Error, style: Lamp-Lamp1-Red
    Label (991,47 154x32), "Robot_Error"
    Label (17,15 365x42), "本界面为电机找零程序："
    Label (83,64 874x42), "可以用来给单个电机或者是整体机器人找零"
    Table (11,121 204x480), data array: Hexapod_Robot.Axis_ActPostion
        p3854506369: Hexapod_Robot.Axis_ActPostion[INDEX]
        p2232123230: Axis_ActPostion[Robot]
    Table (227,122 230x480), data array: Hexapod_Robot.Current_Turque_Value
        p3854506369: Hexapod_Robot.Current_Turque_Value[INDEX]
        p2232123230: Current_Turque_Value[Robot]
    Lamp1 (759,23 61x59), variable: Hexapod_Robot.Robot_Power, style: Lamp-Lamp1-Yellow
    Label (802,47 154x32), "Robot_Power"
    Rectangle (465,121 274x80)
    Button (473,165 80x30), "Axis1_Home"
        toggle Hexapod_Robot.Axis_Home_Set[1]
        OnMouseClick: change screen: Visu_Home
    Button (650,165 80x30), "Axis3_Home"
        toggle Hexapod_Robot.Axis_Home_Set[3]
        OnMouseClick: change screen: Visu_Home
    Button (562,165 80x30), "Axis2_Home"
        toggle Hexapod_Robot.Axis_Home_Set[2]
        OnMouseClick: change screen: Visu_Home
    Rectangle (465,201 274x80)
    Button (473,245 80x30), "Axis4_Home"
        toggle Hexapod_Robot.Axis_Home_Set[4]
        OnMouseClick: change screen: Visu_Home
    Button (650,245 80x30), "Axis6_Home"
        toggle Hexapod_Robot.Axis_Home_Set[6]
        OnMouseClick: change screen: Visu_Home
    Button (562,245 80x30), "Axis5_Home"
        toggle Hexapod_Robot.Axis_Home_Set[5]
        OnMouseClick: change screen: Visu_Home
    Rectangle (465,281 274x80)
    Button (473,325 80x30), "Axis7_Home"
        toggle Hexapod_Robot.Axis_Home_Set[7]
        OnMouseClick: change screen: Visu_Home
    Button (650,325 80x30), "Axis9_Home"
        toggle Hexapod_Robot.Axis_Home_Set[9]
        OnMouseClick: change screen: Visu_Home
    Button (562,325 80x30), "Axis8_Home"
        toggle Hexapod_Robot.Axis_Home_Set[8]
        OnMouseClick: change screen: Visu_Home
    Rectangle (465,361 274x80)
    Button (473,405 80x30), "Axis10_Home"
        toggle Hexapod_Robot.Axis_Home_Set[10]
        OnMouseClick: change screen: Visu_Home
    Button (650,405 80x30), "Axis12_Home"
        toggle Hexapod_Robot.Axis_Home_Set[12]
        OnMouseClick: change screen: Visu_Home
    Button (562,405 80x30), "Axis11_Home"
        toggle Hexapod_Robot.Axis_Home_Set[11]
        OnMouseClick: change screen: Visu_Home
    Rectangle (465,441 274x80)
    Button (473,485 80x30), "Axis13_Home"
        toggle Hexapod_Robot.Axis_Home_Set[13]
        OnMouseClick: change screen: Visu_Home
    Button (650,485 80x30), "Axis15_Home"
        toggle Hexapod_Robot.Axis_Home_Set[15]
        OnMouseClick: change screen: Visu_Home
    Button (562,485 80x30), "Axis14_Home"
        toggle Hexapod_Robot.Axis_Home_Set[14]
        OnMouseClick: change screen: Visu_Home
    Rectangle (465,521 274x80)
    Button (473,565 80x30), "Axis16_Home"
        toggle Hexapod_Robot.Axis_Home_Set[16]
        OnMouseClick: change screen: Visu_Home
    Button (650,565 80x30), "Axis18_Home"
        toggle Hexapod_Robot.Axis_Home_Set[18]
        OnMouseClick: change screen: Visu_Home
    Button (562,565 80x30), "Axis17_Home"
        toggle Hexapod_Robot.Axis_Home_Set[17]
        OnMouseClick: change screen: Visu_Home
    Rectangle (749,498 376x96)
    Rectangle (766,480 182x41), "切换视图"
    Button (762,543 110x43), "Power"
        OnMouseClick: change screen: Visu_Power
    Button (1002,543 110x43), "Error & Reset"
        OnMouseClick: change screen: Visu_Reset
    Button (882,543 110x43), "Simulink_Move"
        OnMouseClick: change screen: Visu_SimulinkMove
    Rectangle (748,122 376x157)
    Rectangle (765,104 182x41), "是否进行整机操作"
    Lamp1 (980,173 80x80), variable: Hexapod_Robot.Robot_Home_Set, style: Lamp-Lamp1-Green
    RotarySwitch (809,173 80x80), variable: Hexapod_Robot.Robot_Home_Set, behaviour: TOGGLE, style: Switch-RotarySwitch-Gray
    Label (864,166 60x30), "否"
    Label (769,166 60x30), "是"
    Label (935,127 207x32), "Robot_Home_Set"
    Button (518,127 150x30), "Leg1_Home"
        tap Hexapod_Robot.Leg_Home_Set[1]
    Button (518,208 150x30), "Leg2_Home"
        tap Hexapod_Robot.Leg_Home_Set[2]
    Button (518,288 150x30), "Leg3_Home"
        tap Hexapod_Robot.Leg_Home_Set[3]
    Button (518,367 150x30), "Leg4_Home"
        tap Hexapod_Robot.Leg_Home_Set[4]
    Button (518,448 150x30), "Leg5_Home"
        tap Hexapod_Robot.Leg_Home_Set[5]
    Button (518,527 150x30), "Leg6_Home"
        tap Hexapod_Robot.Leg_Home_Set[6]
END_VISUALIZATION

// ---- VISUs/Visu_SimulinkMove.TcVIS
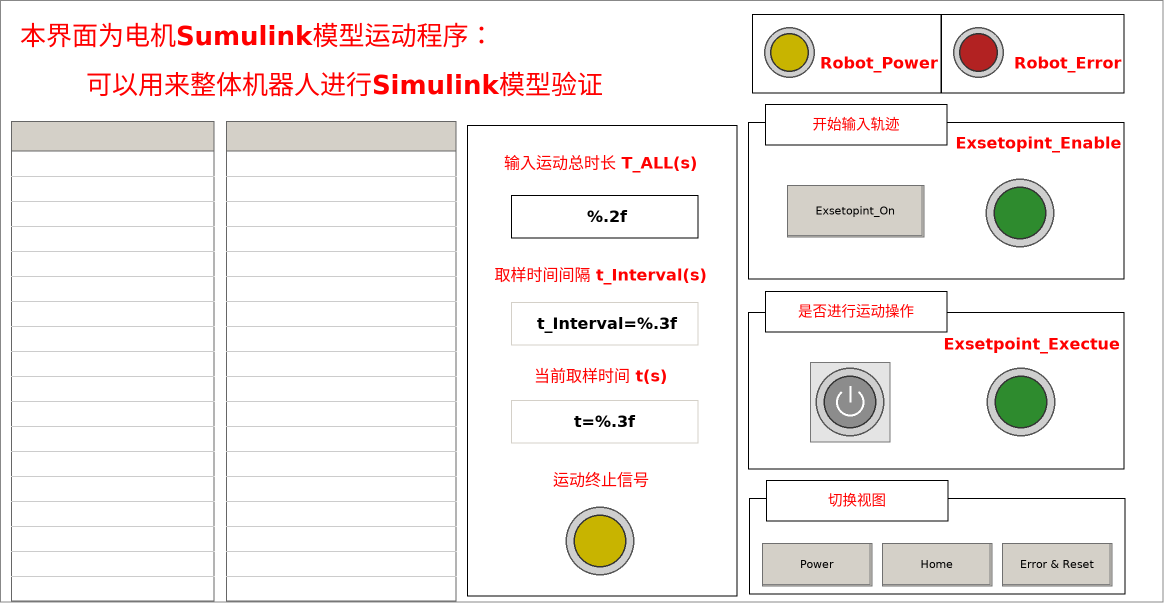
VISUALIZATION Visu_SimulinkMove  // 1164x603
    Rectangle (749,498 376x96)
    Rectangle (766,480 182x41), "切换视图"
    Button (762,543 110x43), "Power"
        OnMouseClick: change screen: Visu_Power
    Button (1002,543 110x43), "Error & Reset"
        OnMouseClick: change screen: Visu_Reset
    Button (882,543 110x43), "Home"
        OnMouseClick: change screen: Visu_Home
    Rectangle (467,125 270x471)
    Rectangle (752,14 189x79)
    Rectangle (748,312 376x157)
    Label (902,328 260x32), "Exsetpoint_Exectue"
    Rectangle (765,291 182x41), "是否进行运动操作"
    Lamp1 (981,362 80x80), variable: ExSetPoint_Execute, style: Lamp-Lamp1-Green
    PowerSwitch (810,362 80x80), variable: ExSetPoint_Execute, behaviour: TOGGLE, style: Switch-PowerSwitch-Gray
    Rectangle (941,14 183x79)
    Lamp1 (948,23 61x59), variable: Hexapod_Robot.Robot_Error, style: Lamp-Lamp1-Red
    Label (991,47 154x32), "Robot_Error"
    Label (17,15 572x42), "本界面为电机Sumulink模型运动程序："
    Label (83,64 874x42), "可以用来整体机器人进行Simulink模型验证"
    Table (11,121 203x480), data array: Hexapod_Robot.Axis_ActPostion
        p3854506369: Hexapod_Robot.Axis_ActPostion[INDEX]
        p2232123230: Axis_ActPostion[Robot]
    Table (226,121 230x480), data array: Hexapod_Robot.Current_Turque_Value
        p3854506369: Hexapod_Robot.Current_Turque_Value[INDEX]
        p2232123230: Current_Turque_Value[Robot]
    Lamp1 (759,23 61x59), variable: Hexapod_Robot.Robot_Power, style: Lamp-Lamp1-Yellow
    Label (802,47 154x32), "Robot_Power"
    Rectangle (748,122 376x157)
    Rectangle (765,104 182x41), "开始输入轨迹"
    Lamp1 (980,173 80x80), variable: MAIN.ExtSetPointEnable, style: Lamp-Lamp1-Green
    Label (935,127 207x32), "Exsetopint_Enable"
    Rectangle (511,195 187x43), "%.2f", text variable: MAIN.T_All
        OnMouseClick: write MAIN.T_All via Default
    Label (471,147 260x32), "输入运动总时长 T_ALL(s)"
    Textfield (511,400 187x43), "t=%.3f", text variable: MAIN.t
    Label (471,360 260x32), "当前取样时间 t(s)"
    Button (787,185 137x52), "Exsetopint_On"
        toggle MAIN.ExtSetPointEnable
    Lamp1 (560,501 80x80), variable: MAIN.ExtSetPointDisable, style: Lamp-Lamp1-Yellow
    Label (471,464 260x32), "运动终止信号"
    Label (471,259 260x32), "取样时间间隔 t_Interval(s)"
    Textfield (511,302 187x43), "t_Interval=%.3f", text variable: MAIN.t_Interval
        OnMouseClick: write MAIN.t_Interval via Default
END_VISUALIZATION

// ---- VISUs/Visu_Power.TcVIS
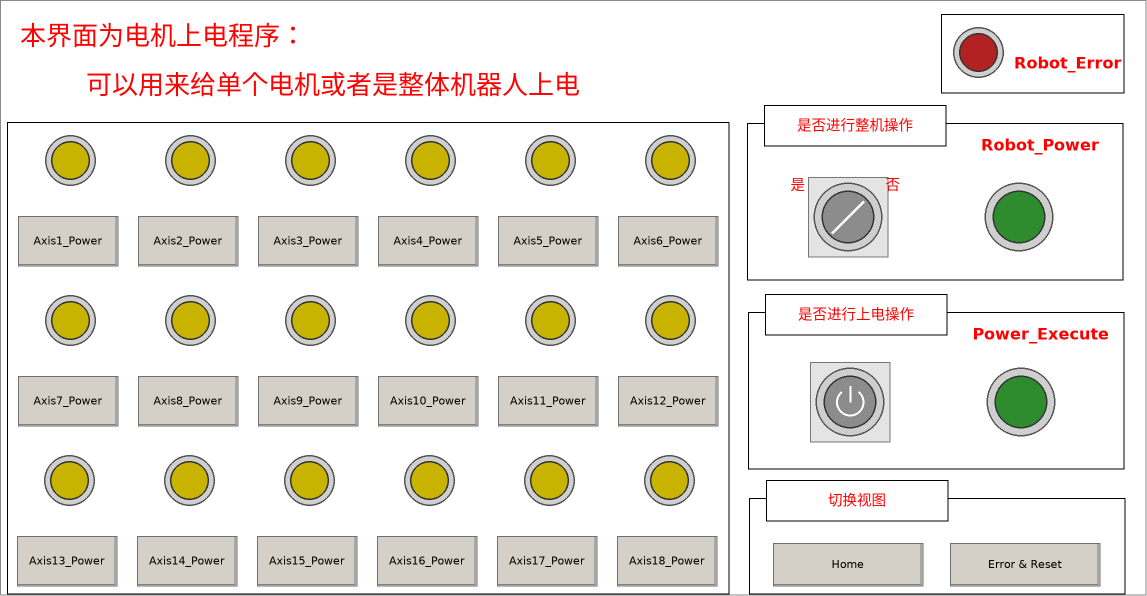
VISUALIZATION Visu_Power  // 1147x596
    Label (987,37 154x32), "Robot_Error"
    Rectangle (7,122 722x472)
    Lamp1 (40,131 61x59), variable: Hexapod_Robot.Power_Status[1], style: Lamp-Lamp1-Yellow
    Lamp1 (160,131 61x59), variable: Hexapod_Robot.Power_Status[2], style: Lamp-Lamp1-Yellow
    Lamp1 (280,131 61x59), variable: Hexapod_Robot.Power_Status[3], style: Lamp-Lamp1-Yellow
    Lamp1 (400,131 61x59), variable: Hexapod_Robot.Power_Status[4], style: Lamp-Lamp1-Yellow
    Lamp1 (520,131 61x59), variable: Hexapod_Robot.Power_Status[5], style: Lamp-Lamp1-Yellow
    Lamp1 (640,131 61x59), variable: Hexapod_Robot.Power_Status[6], style: Lamp-Lamp1-Yellow
    Button (18,216 100x50), "Axis1_Power"
        toggle Hexapod_Robot.Axis_Power[1]
    Button (138,216 100x50), "Axis2_Power"
        toggle Hexapod_Robot.Axis_Power[2]
    Button (258,216 100x50), "Axis3_Power"
        toggle Hexapod_Robot.Axis_Power[3]
    Button (378,216 100x50), "Axis4_Power"
        toggle Hexapod_Robot.Axis_Power[4]
    Button (498,216 100x50), "Axis5_Power"
        toggle Hexapod_Robot.Axis_Power[5]
    Button (618,216 100x50), "Axis6_Power"
        toggle Hexapod_Robot.Axis_Power[6]
    Lamp1 (40,291 61x59), variable: Hexapod_Robot.Power_Status[7], style: Lamp-Lamp1-Yellow
    Lamp1 (160,291 61x59), variable: Hexapod_Robot.Power_Status[8], style: Lamp-Lamp1-Yellow
    Lamp1 (280,291 61x59), variable: Hexapod_Robot.Power_Status[9], style: Lamp-Lamp1-Yellow
    Lamp1 (400,291 61x59), variable: Hexapod_Robot.Power_Status[10], style: Lamp-Lamp1-Yellow
    Lamp1 (520,291 61x59), variable: Hexapod_Robot.Power_Status[11], style: Lamp-Lamp1-Yellow
    Lamp1 (640,291 61x59), variable: Hexapod_Robot.Power_Status[12], style: Lamp-Lamp1-Yellow
    Button (18,376 100x50), "Axis7_Power"
        toggle Hexapod_Robot.Axis_Power[7]
    Button (138,376 100x50), "Axis8_Power"
        toggle Hexapod_Robot.Axis_Power[8]
    Button (258,376 100x50), "Axis9_Power"
        toggle Hexapod_Robot.Axis_Power[9]
    Button (378,376 100x50), "Axis10_Power"
        toggle Hexapod_Robot.Axis_Power[10]
    Button (498,376 100x50), "Axis11_Power"
        toggle Hexapod_Robot.Axis_Power[11]
    Button (618,376 100x50), "Axis12_Power"
        toggle Hexapod_Robot.Axis_Power[12]
    Lamp1 (39,451 61x59), variable: Hexapod_Robot.Power_Status[13], style: Lamp-Lamp1-Yellow
    Lamp1 (159,451 61x59), variable: Hexapod_Robot.Power_Status[14], style: Lamp-Lamp1-Yellow
    Lamp1 (279,451 61x59), variable: Hexapod_Robot.Power_Status[15], style: Lamp-Lamp1-Yellow
    Lamp1 (399,451 61x59), variable: Hexapod_Robot.Power_Status[16], style: Lamp-Lamp1-Yellow
    Lamp1 (519,451 61x59), variable: Hexapod_Robot.Power_Status[17], style: Lamp-Lamp1-Yellow
    Lamp1 (639,451 61x59), variable: Hexapod_Robot.Power_Status[18], style: Lamp-Lamp1-Yellow
    Button (17,536 100x50), "Axis13_Power"
        toggle Hexapod_Robot.Axis_Power[13]
    Button (137,536 100x50), "Axis14_Power"
        toggle Hexapod_Robot.Axis_Power[14]
    Button (257,536 100x50), "Axis15_Power"
        toggle Hexapod_Robot.Axis_Power[15]
    Button (377,536 100x50), "Axis16_Power"
        toggle Hexapod_Robot.Axis_Power[16]
    Button (497,536 100x50), "Axis17_Power"
        toggle Hexapod_Robot.Axis_Power[17]
    Button (617,536 100x50), "Axis18_Power"
        toggle Hexapod_Robot.Axis_Power[18]
    Rectangle (748,312 376x157)
    Label (964,318 154x32), "Power_Execute"
    Rectangle (765,294 182x41), "是否进行上电操作"
    Lamp1 (981,362 80x80), variable: Power_Execute, style: Lamp-Lamp1-Green
    Rectangle (749,498 376x96)
    Rectangle (766,480 182x41), "切换视图"
    Button (773,543 150x43), "Home"
        OnMouseClick: change screen: Visu_Home
    PowerSwitch (810,362 80x80), variable: Power_Execute, behaviour: TOGGLE, style: Switch-PowerSwitch-Gray
    Rectangle (941,14 183x79)
    Lamp1 (948,23 61x59), variable: Hexapod_Robot.Robot_Error, style: Lamp-Lamp1-Red
    Label (17,15 365x42), "本界面为电机上电程序："
    Label (83,64 639x42), "可以用来给单个电机或者是整体机器人上电"
    Button (950,543 150x43), "Error & Reset"
        OnMouseClick: change screen: Visu_Reset
    Rectangle (747,123 376x157)
    Label (963,129 154x32), "Robot_Power"
    Rectangle (764,105 182x41), "是否进行整机操作"
    Lamp1 (979,177 80x80), variable: Hexapod_Robot.Robot_Power, style: Lamp-Lamp1-Green
    RotarySwitch (808,177 80x80), variable: Hexapod_Robot.Robot_Power, behaviour: TOGGLE, style: Switch-RotarySwitch-Gray
    Label (863,170 60x30), "否"
    Label (768,170 60x30), "是"
    Label (991,47 154x32), "Robot_Error"
END_VISUALIZATION

// ---- VISUs/Visu_Reset.TcVIS
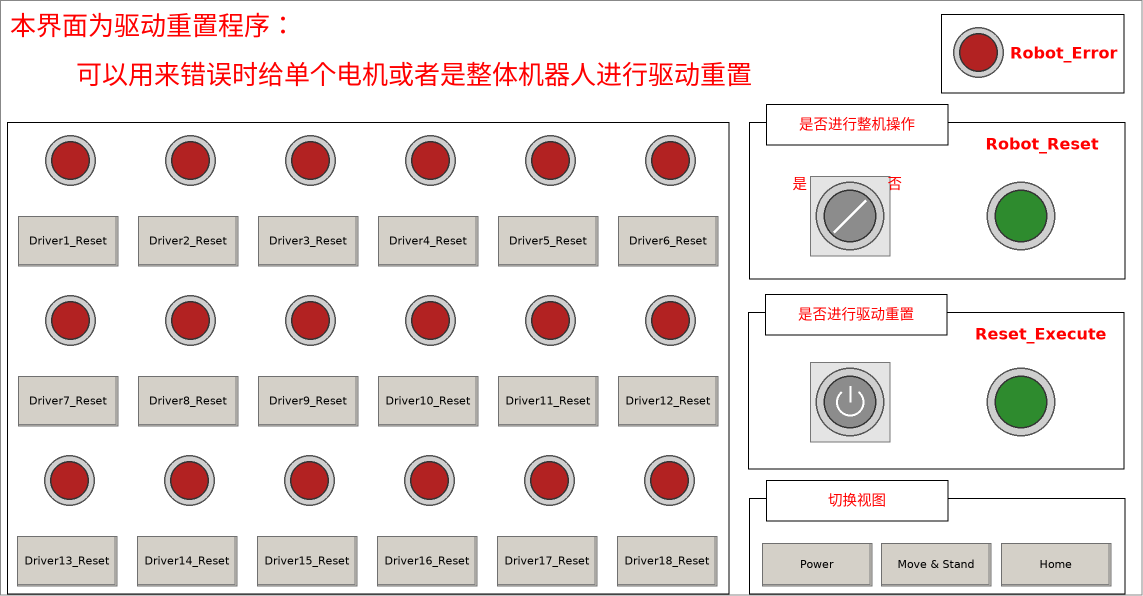
VISUALIZATION Visu_Reset  // 1143x596
    Rectangle (7,122 722x472)
    Lamp1 (40,131 61x59), variable: Hexapod_Robot.Axis_Error[1], style: Lamp-Lamp1-Red
    Lamp1 (160,131 61x59), variable: Hexapod_Robot.Axis_Error[2], style: Lamp-Lamp1-Red
    Lamp1 (280,131 61x59), variable: Hexapod_Robot.Axis_Error[3], style: Lamp-Lamp1-Red
    Lamp1 (400,131 61x59), variable: Hexapod_Robot.Axis_Error[4], style: Lamp-Lamp1-Red
    Lamp1 (520,131 61x59), variable: Hexapod_Robot.Axis_Error[5], style: Lamp-Lamp1-Red
    Lamp1 (640,131 61x59), variable: Hexapod_Robot.Axis_Error[6], style: Lamp-Lamp1-Red
    Button (18,216 100x50), "Driver1_Reset"
        tap Hexapod_Robot.Axis_Reset[1]
    Button (138,216 100x50), "Driver2_Reset"
        tap Hexapod_Robot.Axis_Reset[2]
    Button (258,216 100x50), "Driver3_Reset"
        tap Hexapod_Robot.Axis_Reset[3]
    Button (378,216 100x50), "Driver4_Reset"
        tap Hexapod_Robot.Axis_Reset[4]
    Button (498,216 100x50), "Driver5_Reset"
        tap Hexapod_Robot.Axis_Reset[5]
    Button (618,216 100x50), "Driver6_Reset"
        tap Hexapod_Robot.Axis_Reset[6]
    Lamp1 (40,291 61x59), variable: Hexapod_Robot.Axis_Error[7], style: Lamp-Lamp1-Red
    Lamp1 (160,291 61x59), variable: Hexapod_Robot.Axis_Error[8], style: Lamp-Lamp1-Red
    Lamp1 (280,291 61x59), variable: Hexapod_Robot.Axis_Error[9], style: Lamp-Lamp1-Red
    Lamp1 (400,291 61x59), variable: Hexapod_Robot.Axis_Error[10], style: Lamp-Lamp1-Red
    Lamp1 (520,291 61x59), variable: Hexapod_Robot.Axis_Error[11], style: Lamp-Lamp1-Red
    Lamp1 (640,291 61x59), variable: Hexapod_Robot.Axis_Error[12], style: Lamp-Lamp1-Red
    Button (18,376 100x50), "Driver7_Reset"
        tap Hexapod_Robot.Axis_Reset[7]
    Button (138,376 100x50), "Driver8_Reset"
        tap Hexapod_Robot.Axis_Reset[8]
    Button (258,376 100x50), "Driver9_Reset"
        tap Hexapod_Robot.Axis_Reset[9]
    Button (378,376 100x50), "Driver10_Reset"
        tap Hexapod_Robot.Axis_Reset[10]
    Button (498,376 100x50), "Driver11_Reset"
        tap Hexapod_Robot.Axis_Reset[11]
    Button (618,376 100x50), "Driver12_Reset"
        tap Hexapod_Robot.Axis_Reset[12]
    Lamp1 (39,451 61x59), variable: Hexapod_Robot.Axis_Error[13], style: Lamp-Lamp1-Red
    Lamp1 (159,451 61x59), variable: Hexapod_Robot.Axis_Error[14], style: Lamp-Lamp1-Red
    Lamp1 (279,451 61x59), variable: Hexapod_Robot.Axis_Error[15], style: Lamp-Lamp1-Red
    Lamp1 (399,451 61x59), variable: Hexapod_Robot.Axis_Error[16], style: Lamp-Lamp1-Red
    Lamp1 (519,451 61x59), variable: Hexapod_Robot.Axis_Error[17], style: Lamp-Lamp1-Red
    Lamp1 (639,451 61x59), variable: Hexapod_Robot.Axis_Error[18], style: Lamp-Lamp1-Red
    Button (17,536 100x50), "Driver13_Reset"
        tap Hexapod_Robot.Axis_Reset[13]
    Button (137,536 100x50), "Driver14_Reset"
        tap Hexapod_Robot.Axis_Reset[14]
    Button (257,536 100x50), "Driver15_Reset"
        tap Hexapod_Robot.Axis_Reset[15]
    Button (377,536 100x50), "Driver16_Reset"
        tap Hexapod_Robot.Axis_Reset[16]
    Button (497,536 100x50), "Driver17_Reset"
        tap Hexapod_Robot.Axis_Reset[17]
    Button (617,536 100x50), "Driver18_Reset"
        tap Hexapod_Robot.Axis_Reset[18]
    Rectangle (749,122 376x157)
    Label (965,128 154x32), "Robot_Reset"
    Rectangle (766,104 182x41), "是否进行整机操作"
    Rectangle (748,312 376x157)
    Label (964,318 154x32), "Reset_Execute"
    Rectangle (765,294 182x41), "是否进行驱动重置"
    Lamp1 (981,176 80x80), variable: Hexapod_Robot.Robot_Reset, style: Lamp-Lamp1-Green
    Lamp1 (981,362 80x80), variable: Reset_Execute, style: Lamp-Lamp1-Green
    RotarySwitch (810,176 80x80), variable: Hexapod_Robot.Robot_Reset, behaviour: TOGGLE, style: Switch-RotarySwitch-Gray
    Rectangle (749,498 376x96)
    Rectangle (766,480 182x41), "切换视图"
    Label (865,169 60x30), "否"
    Label (770,169 60x30), "是"
    PowerSwitch (810,362 80x80), variable: Reset_Execute, behaviour: TOGGLE, style: Switch-PowerSwitch-Gray
    Label (7,5 365x42), "本界面为驱动重置程序："
    Label (73,54 874x42), "可以用来错误时给单个电机或者是整体机器人进行驱动重置"
    Rectangle (941,14 183x79)
    Lamp1 (948,23 61x59), variable: Hexapod_Robot.Robot_Error, style: Lamp-Lamp1-Red
    Label (987,37 154x32), "Robot_Error"
    Button (762,543 110x43), "Power"
        OnMouseClick: change screen: Visu_Power
    Button (1001,543 110x43), "Home"
        OnMouseClick: change screen: Visu_Home
    Button (881,543 110x43), "Move & Stand"
        OnMouseClick: change screen: Visu_Stand
END_VISUALIZATION
